SPLINE
SPL {X  -162.820, Y  +507.703, Z    +0.000, E1   -49.462, E3 +312953.270}
SPL {X  -162.820, Y  +516.435, Z    +0.000, E1   -49.526, E3 +312968.239}
SPL {X  -162.820, Y  +523.383, Z    +0.000, E1   -49.407, E3 +312981.426}
SPL {X  -162.820, Y  +532.283, Z    +0.000, E1   -49.462, E3 +312997.028}
SPL {X  -162.820, Y  +541.471, Z    +0.000, E1   -49.456, E3 +313013.407}
SPL {X  -162.820, Y  +548.933, Z    +0.000, E1   -49.456, E3 +313026.595}
SPL {X  -162.820, Y  +553.997, Z    +0.000, E1   -49.325, E3 +313036.399}
SPL {X  -162.820, Y  +562.346, Z    +0.000, E1   -49.498, E3 +313050.461}
SPL {X  -162.820, Y  +570.444, Z    +0.000, E1   -49.421, E3 +313065.208}
SPL {X  -162.820, Y  +577.429, Z    +0.000, E1   -49.474, E3 +313077.322}
SPL {X  -162.820, Y  +585.965, Z    +0.000, E1   -49.447, E3 +313092.896}
SPL {X  -162.820, Y  +594.192, Z    +0.000, E1   -49.325, E3 +313108.139}
SPL {X  -162.820, Y  +600.267, Z    +0.000, E1   -49.443, E3 +313118.228}
SPL {X  -162.820, Y  +606.218, Z    +0.000, E1   -49.464, E3 +313128.775}
SPL {X  -162.820, Y  +612.538, Z    +0.000, E1   -49.488, E3 +313139.826}
SPL {X  -162.820, Y  +617.738, Z    +0.000, E1   -49.301, E3 +313150.262}
SPL {X  -162.820, Y  +624.265, Z    +0.000, E1   -49.443, E3 +313161.057}
SPL {X  -162.820, Y  +630.226, Z    +0.000, E1   -49.472, E3 +313171.505}
SPL {X  -162.820, Y  +635.239, Z    +0.000, E1   -49.373, E3 +313181.001}
SPL {X  -162.820, Y  +641.207, Z    +0.000, E1   -49.420, E3 +313191.469}
SPL {X  -162.820, Y  +649.864, Z    +0.000, E1   -49.433, E3 +313206.947}
SPL {X  -162.820, Y  +658.147, Z    +0.000, E1   -49.491, E3 +313221.214}
SPL {X  -162.820, Y  +663.916, Z    +0.000, E1   -49.371, E3 +313232.204}
SPL {X  -162.820, Y  +669.755, Z    +0.000, E1   -49.387, E3 +313242.529}
SPL {X  -162.807, Y  +675.597, Z    +0.000, E1   -49.472, E3 +313252.431}
SPL {X  -162.632, Y  +681.322, Z    +0.000, E1   -49.345, E3 +313263.443}
SPL {X  -162.228, Y  +687.372, Z    +0.000, E1   -49.294, E3 +313274.529}
SPL {X  -161.723, Y  +692.372, Z    +0.000, E1   -49.172, E3 +313284.159}
SPL {X  -161.009, Y  +697.714, Z    +0.000, E1   -49.214, E3 +313293.444}
SPL {X  -160.313, Y  +701.965, Z    +0.000, E1   -48.932, E3 +313302.656}
SPL {X  -158.980, Y  +708.651, Z    +0.000, E1   -48.774, E3 +313315.696}
SPL {X  -157.477, Y  +714.869, Z    +0.000, E1   -48.424, E3 +313328.571}
SPL {X  -156.071, Y  +719.891, Z    +0.000, E1   -48.264, E3 +313338.447}
SPL {X  -154.661, Y  +724.395, Z    +0.000, E1   -47.951, E3 +313348.129}
SPL {X  -153.094, Y  +728.931, Z    +0.000, E1   -47.705, E3 +313357.565}
SPL {X  -151.300, Y  +733.655, Z    +0.000, E1   -47.339, E3 +313367.874}
SPL {X  -145.669, Y  +746.239, Z    +0.000, E1   -50.198, E3 +313374.650}
SPL {X  -135.559, Y  +763.690, Z    +0.000, E1   -44.340, E3 +313461.445}
ENDSPLINE

SPLINE
SPL {X  -153.801, Y  +726.938, Z    +0.000, E1   -29.643, E3 +313530.158}
SPL {X  -160.383, Y  +701.564, Z    +0.000, E1   -18.145, E3 +313538.297}
SPL {X  -162.078, Y  +689.023, Z    +0.000, E1   -11.510, E3 +313537.835}
SPL {X  -162.685, Y  +680.136, Z    +0.000, E1    -6.379, E3 +313538.124}
SPL {X  -162.820, Y  +672.919, Z    +0.000, E1    -1.752, E3 +313538.163}
SPL {X  -162.820, Y  +667.861, Z    +0.000, E1    +2.254, E3 +313537.964}
SPL {X  -162.820, Y  +662.755, Z    +0.000, E1    +7.521, E3 +313538.005}
SPL {X  -162.820, Y  +657.537, Z    +0.000, E1   +13.540, E3 +313537.674}
SPL {X  -162.820, Y  +650.460, Z    +0.000, E1   +22.200, E3 +313537.105}
SPL {X  -162.820, Y  +637.843, Z    +0.000, E1   +35.051, E3 +313539.182}
SPL {X  -162.820, Y  +595.072, Z    +0.000, E1   +53.652, E3 +313559.902}
SPL {X  -162.820, Y  +560.706, Z    +0.000, E1   +50.482, E3 +313620.811}
ENDSPLINE

SPLINE
SPL {X  -162.820, Y  +560.978, Z    +0.000, E1   +48.448, E3 +313632.897}
ENDSPLINE

SPLINE
SPL {X  -162.820, Y  +552.125, Z    +0.000, E1   +48.477, E3 +313649.002}
SPL {X  -162.820, Y  +545.800, Z    +0.000, E1   +48.334, E3 +313661.443}
SPL {X  -162.820, Y  +540.645, Z    +0.000, E1   +48.364, E3 +313670.794}
SPL {X  -162.820, Y  +534.689, Z    +0.000, E1   +48.295, E3 +313682.343}
SPL {X  -162.820, Y  +526.053, Z    +0.000, E1   +48.382, E3 +313697.918}
SPL {X  -162.820, Y  +516.130, Z    +0.000, E1   +48.458, E3 +313715.876}
SPL {X  -162.820, Y  +508.282, Z    +0.000, E1   +48.307, E3 +313731.131}
SPL {X  -162.820, Y  +502.890, Z    +0.000, E1   +48.309, E3 +313741.058}
ENDSPLINE

SPLINE
SPL {X  -162.820, Y  +517.326, Z    +0.000, E1   +41.232, E3 +313753.322}
ENDSPLINE

SPLINE
SPL {X  -162.820, Y  +509.871, Z    +0.000, E1   +42.115, E3 +313765.423}
SPL {X  -162.820, Y  +504.481, Z    +0.000, E1   +42.725, E3 +313774.088}
SPL {X  -162.820, Y  +496.780, Z    +0.000, E1   +43.573, E3 +313786.255}
SPL {X  -162.820, Y  +488.962, Z    +0.000, E1   +44.342, E3 +313798.523}
SPL {X  -162.820, Y  +481.373, Z    +0.000, E1   +45.107, E3 +313810.007}
SPL {X  -162.820, Y  +473.909, Z    +0.000, E1   +45.743, E3 +313821.520}
SPL {X  -162.820, Y  +465.836, Z    +0.000, E1   +46.727, E3 +313831.810}
SPL {X  -162.820, Y  +457.217, Z    +0.000, E1   +47.671, E3 +313842.848}
SPL {X  -162.820, Y  +449.104, Z    +0.000, E1   +48.459, E3 +313853.317}
SPL {X  -162.820, Y  +438.072, Z    +0.000, E1   +49.432, E3 +313867.672}
SPL {X  -162.820, Y  +428.488, Z    +0.000, E1   +49.830, E3 +313882.107}
SPL {X  -162.820, Y  +423.062, Z    +0.000, E1   +49.728, E3 +313892.250}
SPL {X  -162.820, Y  +416.560, Z    +0.000, E1   +49.816, E3 +313903.231}
SPL {X  -162.820, Y  +410.559, Z    +0.000, E1   +49.727, E3 +313914.286}
SPL {X  -162.820, Y  +405.170, Z    +0.000, E1   +49.772, E3 +313923.488}
SPL {X  -162.820, Y  +398.766, Z    +0.000, E1   +49.793, E3 +313934.775}
SPL {X  -162.820, Y  +391.831, Z    +0.000, E1   +49.801, E3 +313946.821}
SPL {X  -162.820, Y  +386.334, Z    +0.000, E1   +49.739, E3 +313956.910}
SPL {X  -162.801, Y  +377.981, Z    +0.000, E1   +49.798, E3 +313971.431}
SPL {X  -162.314, Y  +367.677, Z    +0.000, E1   +49.734, E3 +313990.071}
SPL {X  -161.359, Y  +358.734, Z    +0.000, E1   +49.535, E3 +314006.855}
SPL {X  -160.051, Y  +350.597, Z    +0.000, E1   +49.332, E3 +314022.465}
SPL {X  -158.863, Y  +344.823, Z    +0.000, E1   +49.020, E3 +314034.193}
SPL {X  -157.695, Y  +339.971, Z    +0.000, E1   +48.934, E3 +314043.289}
SPL {X  -156.136, Y  +334.326, Z    +0.000, E1   +48.578, E3 +314055.256}
SPL {X  -154.561, Y  +329.302, Z    +0.000, E1   +48.290, E3 +314065.586}
SPL {X  -152.787, Y  +324.229, Z    +0.000, E1   +47.981, E3 +314076.276}
SPL {X  -150.789, Y  +319.074, Z    +0.000, E1   +47.585, E3 +314087.299}
SPL {X  -145.123, Y  +306.679, Z    +0.000, E1   +50.518, E3 +314093.196}
SPL {X  -135.207, Y  +289.783, Z    +0.000, E1   +44.101, E3 +314186.711}
ENDSPLINE

SPLINE
SPL {X  -154.528, Y  +329.203, Z    +0.000, E1   +28.834, E3 +314257.072}
SPL {X  -160.380, Y  +352.419, Z    +0.000, E1   +18.163, E3 +314261.432}
SPL {X  -162.408, Y  +368.921, Z    +0.000, E1    +9.337, E3 +314260.182}
SPL {X  -162.817, Y  +379.558, Z    +0.000, E1    +2.744, E3 +314260.572}
SPL {X  -162.820, Y  +383.077, Z    +0.000, E1    +0.110, E3 +314260.968}
SPL {X  -162.820, Y  +386.028, Z    +0.000, E1    -2.328, E3 +314260.291}
SPL {X  -162.820, Y  +389.792, Z    +0.000, E1    -6.211, E3 +314260.223}
SPL {X  -162.820, Y  +394.068, Z    +0.000, E1   -11.043, E3 +314260.340}
SPL {X  -162.820, Y  +398.921, Z    +0.000, E1   -16.945, E3 +314260.393}
SPL {X  -162.820, Y  +406.317, Z    +0.000, E1   -26.128, E3 +314259.206}
SPL {X  -162.820, Y  +413.297, Z    +0.000, E1   -33.931, E3 +314259.195}
SPL {X  -162.820, Y  +446.299, Z    +0.000, E1   -49.360, E3 +314279.705}
SPL {X  -162.820, Y  +502.427, Z    +0.000, E1   -53.345, E3 +314342.691}
ENDSPLINE

SPLINE
SPL {X  -162.820, Y  +494.458, Z    +0.000, E1   -49.332, E3 +314353.223}
ENDSPLINE

SPLINE
SPL {X  -162.820, Y  +499.429, Z    +0.000, E1   -49.453, E3 +314361.432}
SPL {X  -162.820, Y  +507.703, Z    +0.000, E1   -49.462, E3 +314376.347}
SPL {X  -162.820, Y  +516.435, Z    +0.000, E1   -49.526, E3 +314391.316}
SPL {X  -162.820, Y  +522.095, Z    +0.000, E1   -49.420, E3 +314402.013}
SPL {X  -162.820, Y  +529.397, Z    +0.000, E1   -49.440, E3 +314415.021}
SPL {X  -162.820, Y  +535.099, Z    +0.000, E1   -49.339, E3 +314425.639}
SPL {X  -162.820, Y  +541.471, Z    +0.000, E1   -49.456, E3 +314436.484}
SPL {X  -162.820, Y  +548.933, Z    +0.000, E1   -49.456, E3 +314449.672}
SPL {X  -162.820, Y  +553.997, Z    +0.000, E1   -49.325, E3 +314459.476}
SPL {X  -162.820, Y  +560.268, Z    +0.000, E1   -49.531, E3 +314469.434}
SPL {X  -162.820, Y  +564.590, Z    +0.000, E1   -49.361, E3 +314478.133}
SPL {X  -162.820, Y  +570.444, Z    +0.000, E1   -49.421, E3 +314488.285}
SPL {X  -162.820, Y  +577.429, Z    +0.000, E1   -49.474, E3 +314500.399}
SPL {X  -162.820, Y  +582.387, Z    +0.000, E1   -49.269, E3 +314510.420}
SPL {X  -162.820, Y  +588.456, Z    +0.000, E1   -49.496, E3 +314519.935}
SPL {X  -162.820, Y  +594.192, Z    +0.000, E1   -49.325, E3 +314531.216}
SPL {X  -162.820, Y  +600.267, Z    +0.000, E1   -49.443, E3 +314541.305}
SPL {X  -162.820, Y  +606.218, Z    +0.000, E1   -49.464, E3 +314551.851}
SPL {X  -162.820, Y  +612.538, Z    +0.000, E1   -49.488, E3 +314562.902}
SPL {X  -162.820, Y  +617.738, Z    +0.000, E1   -49.301, E3 +314573.339}
SPL {X  -162.820, Y  +624.265, Z    +0.000, E1   -49.443, E3 +314584.134}
SPL {X  -162.820, Y  +630.226, Z    +0.000, E1   -49.472, E3 +314594.582}
SPL {X  -162.820, Y  +635.239, Z    +0.000, E1   -49.373, E3 +314604.077}
SPL {X  -162.820, Y  +641.207, Z    +0.000, E1   -49.420, E3 +314614.546}
SPL {X  -162.820, Y  +649.864, Z    +0.000, E1   -49.433, E3 +314630.024}
SPL {X  -162.820, Y  +658.147, Z    +0.000, E1   -49.491, E3 +314644.291}
SPL {X  -162.820, Y  +663.916, Z    +0.000, E1   -49.371, E3 +314655.281}
SPL {X  -162.820, Y  +669.755, Z    +0.000, E1   -49.387, E3 +314665.606}
SPL {X  -162.807, Y  +675.597, Z    +0.000, E1   -49.472, E3 +314675.508}
SPL {X  -162.632, Y  +681.322, Z    +0.000, E1   -49.345, E3 +314686.520}
SPL {X  -162.228, Y  +687.372, Z    +0.000, E1   -49.294, E3 +314697.606}
SPL {X  -161.723, Y  +692.372, Z    +0.000, E1   -49.172, E3 +314707.236}
SPL {X  -161.009, Y  +697.714, Z    +0.000, E1   -49.214, E3 +314716.521}
SPL {X  -160.313, Y  +701.965, Z    +0.000, E1   -48.932, E3 +314725.733}
SPL {X  -158.980, Y  +708.651, Z    +0.000, E1   -48.774, E3 +314738.773}
SPL {X  -157.477, Y  +714.869, Z    +0.000, E1   -48.424, E3 +314751.648}
SPL {X  -156.071, Y  +719.891, Z    +0.000, E1   -48.264, E3 +314761.524}
SPL {X  -154.661, Y  +724.395, Z    +0.000, E1   -47.951, E3 +314771.206}
SPL {X  -153.094, Y  +728.931, Z    +0.000, E1   -47.705, E3 +314780.642}
SPL {X  -151.300, Y  +733.655, Z    +0.000, E1   -47.339, E3 +314790.951}
SPL {X  -145.669, Y  +746.239, Z    +0.000, E1   -50.198, E3 +314797.727}
SPL {X  -135.084, Y  +764.399, Z    +0.000, E1   -44.787, E3 +314880.631}
ENDSPLINE

SPLINE
SPL {X  -153.038, Y  +729.086, Z    +0.000, E1   -30.522, E3 +314951.338}
SPL {X  -160.383, Y  +701.564, Z    +0.000, E1   -18.145, E3 +314961.374}
SPL {X  -162.078, Y  +689.023, Z    +0.000, E1   -11.510, E3 +314960.912}
SPL {X  -162.685, Y  +680.136, Z    +0.000, E1    -6.379, E3 +314961.201}
SPL {X  -162.820, Y  +672.919, Z    +0.000, E1    -1.752, E3 +314961.240}
SPL {X  -162.820, Y  +667.861, Z    +0.000, E1    +2.254, E3 +314961.041}
SPL {X  -162.820, Y  +662.755, Z    +0.000, E1    +7.521, E3 +314961.082}
SPL {X  -162.820, Y  +657.537, Z    +0.000, E1   +13.540, E3 +314960.751}
SPL {X  -162.820, Y  +650.460, Z    +0.000, E1   +22.200, E3 +314960.182}
SPL {X  -162.820, Y  +637.843, Z    +0.000, E1   +35.051, E3 +314962.259}
SPL {X  -162.820, Y  +595.072, Z    +0.000, E1   +53.652, E3 +314982.979}
SPL {X  -162.820, Y  +560.706, Z    +0.000, E1   +50.482, E3 +315043.888}
ENDSPLINE

SPLINE
SPL {X  -162.820, Y  +560.978, Z    +0.000, E1   +48.448, E3 +315055.974}
ENDSPLINE

SPLINE
SPL {X  -162.820, Y  +552.125, Z    +0.000, E1   +48.477, E3 +315072.078}
SPL {X  -162.820, Y  +545.800, Z    +0.000, E1   +48.334, E3 +315084.520}
SPL {X  -162.820, Y  +540.645, Z    +0.000, E1   +48.364, E3 +315093.871}
SPL {X  -162.820, Y  +534.689, Z    +0.000, E1   +48.295, E3 +315105.420}
SPL {X  -162.820, Y  +526.053, Z    +0.000, E1   +48.382, E3 +315120.995}
SPL {X  -162.820, Y  +516.130, Z    +0.000, E1   +48.458, E3 +315138.953}
SPL {X  -162.820, Y  +508.282, Z    +0.000, E1   +48.307, E3 +315154.208}
SPL {X  -162.820, Y  +502.890, Z    +0.000, E1   +48.309, E3 +315164.135}
ENDSPLINE

SPLINE
SPL {X  -162.820, Y  +517.326, Z    +0.000, E1   +41.232, E3 +315176.399}
ENDSPLINE

SPLINE
SPL {X  -162.820, Y  +509.871, Z    +0.000, E1   +42.115, E3 +315188.500}
SPL {X  -162.820, Y  +504.481, Z    +0.000, E1   +42.725, E3 +315197.165}
SPL {X  -162.820, Y  +496.780, Z    +0.000, E1   +43.573, E3 +315209.332}
SPL {X  -162.820, Y  +488.962, Z    +0.000, E1   +44.342, E3 +315221.600}
SPL {X  -162.820, Y  +481.373, Z    +0.000, E1   +45.107, E3 +315233.084}
SPL {X  -162.820, Y  +473.909, Z    +0.000, E1   +45.743, E3 +315244.596}
SPL {X  -162.820, Y  +465.836, Z    +0.000, E1   +46.727, E3 +315254.887}
SPL {X  -162.820, Y  +457.217, Z    +0.000, E1   +47.671, E3 +315265.925}
SPL {X  -162.820, Y  +449.104, Z    +0.000, E1   +48.459, E3 +315276.394}
SPL {X  -162.820, Y  +438.072, Z    +0.000, E1   +49.432, E3 +315290.749}
SPL {X  -162.820, Y  +428.488, Z    +0.000, E1   +49.830, E3 +315305.184}
SPL {X  -162.820, Y  +423.062, Z    +0.000, E1   +49.728, E3 +315315.327}
SPL {X  -162.820, Y  +416.560, Z    +0.000, E1   +49.816, E3 +315326.307}
SPL {X  -162.820, Y  +410.559, Z    +0.000, E1   +49.727, E3 +315337.363}
SPL {X  -162.820, Y  +405.170, Z    +0.000, E1   +49.772, E3 +315346.565}
SPL {X  -162.820, Y  +398.766, Z    +0.000, E1   +49.793, E3 +315357.852}
SPL {X  -162.820, Y  +391.831, Z    +0.000, E1   +49.801, E3 +315369.898}
SPL {X  -162.820, Y  +386.334, Z    +0.000, E1   +49.739, E3 +315379.986}
SPL {X  -162.801, Y  +377.981, Z    +0.000, E1   +49.798, E3 +315394.508}
SPL {X  -162.314, Y  +367.677, Z    +0.000, E1   +49.734, E3 +315413.148}
SPL {X  -161.359, Y  +358.734, Z    +0.000, E1   +49.535, E3 +315429.932}
SPL {X  -160.051, Y  +350.597, Z    +0.000, E1   +49.332, E3 +315445.542}
SPL {X  -158.863, Y  +344.823, Z    +0.000, E1   +49.020, E3 +315457.270}
SPL {X  -157.695, Y  +339.971, Z    +0.000, E1   +48.934, E3 +315466.366}
SPL {X  -156.136, Y  +334.326, Z    +0.000, E1   +48.578, E3 +315478.332}
SPL {X  -154.561, Y  +329.302, Z    +0.000, E1   +48.290, E3 +315488.663}
SPL {X  -152.787, Y  +324.229, Z    +0.000, E1   +47.981, E3 +315499.353}
SPL {X  -150.789, Y  +319.074, Z    +0.000, E1   +47.585, E3 +315510.376}
SPL {X  -145.123, Y  +306.679, Z    +0.000, E1   +50.518, E3 +315516.273}
SPL {X  -135.207, Y  +289.783, Z    +0.000, E1   +44.101, E3 +315609.788}
ENDSPLINE

SPLINE
SPL {X  -154.528, Y  +329.203, Z    +0.000, E1   +28.834, E3 +315680.149}
SPL {X  -160.380, Y  +352.419, Z    +0.000, E1   +18.163, E3 +315684.509}
SPL {X  -162.408, Y  +368.921, Z    +0.000, E1    +9.337, E3 +315683.259}
SPL {X  -162.817, Y  +379.558, Z    +0.000, E1    +2.744, E3 +315683.649}
SPL {X  -162.820, Y  +383.077, Z    +0.000, E1    +0.110, E3 +315684.045}
SPL {X  -162.820, Y  +386.028, Z    +0.000, E1    -2.328, E3 +315683.368}
SPL {X  -162.820, Y  +389.792, Z    +0.000, E1    -6.211, E3 +315683.300}
SPL {X  -162.820, Y  +394.068, Z    +0.000, E1   -11.043, E3 +315683.417}
SPL {X  -162.820, Y  +398.921, Z    +0.000, E1   -16.945, E3 +315683.470}
SPL {X  -162.820, Y  +406.317, Z    +0.000, E1   -26.128, E3 +315682.283}
SPL {X  -162.820, Y  +413.297, Z    +0.000, E1   -33.931, E3 +315682.272}
SPL {X  -162.820, Y  +446.299, Z    +0.000, E1   -49.360, E3 +315702.782}
SPL {X  -162.820, Y  +502.427, Z    +0.000, E1   -53.345, E3 +315765.768}
ENDSPLINE

SPLINE
SPL {X  -162.820, Y  +494.458, Z    +0.000, E1   -49.332, E3 +315776.300}
ENDSPLINE

SPLINE
SPL {X  -162.820, Y  +499.429, Z    +0.000, E1   -49.453, E3 +315784.509}
SPL {X  -162.820, Y  +507.703, Z    +0.000, E1   -49.462, E3 +315799.424}
SPL {X  -162.820, Y  +516.435, Z    +0.000, E1   -49.526, E3 +315814.393}
SPL {X  -162.820, Y  +522.095, Z    +0.000, E1   -49.420, E3 +315825.090}
SPL {X  -162.820, Y  +529.397, Z    +0.000, E1   -49.440, E3 +315838.098}
SPL {X  -162.820, Y  +535.099, Z    +0.000, E1   -49.339, E3 +315848.716}
SPL {X  -162.820, Y  +541.471, Z    +0.000, E1   -49.456, E3 +315859.560}
SPL {X  -162.820, Y  +548.933, Z    +0.000, E1   -49.456, E3 +315872.749}
SPL {X  -162.820, Y  +553.997, Z    +0.000, E1   -49.325, E3 +315882.553}
SPL {X  -162.820, Y  +560.268, Z    +0.000, E1   -49.531, E3 +315892.511}
SPL {X  -162.820, Y  +564.590, Z    +0.000, E1   -49.361, E3 +315901.210}
SPL {X  -162.820, Y  +570.444, Z    +0.000, E1   -49.421, E3 +315911.362}
SPL {X  -162.820, Y  +577.429, Z    +0.000, E1   -49.474, E3 +315923.476}
SPL {X  -162.820, Y  +582.387, Z    +0.000, E1   -49.269, E3 +315933.497}
SPL {X  -162.820, Y  +588.456, Z    +0.000, E1   -49.496, E3 +315943.012}
SPL {X  -162.820, Y  +594.192, Z    +0.000, E1   -49.325, E3 +315954.293}
SPL {X  -162.820, Y  +600.267, Z    +0.000, E1   -49.443, E3 +315964.382}
SPL {X  -162.820, Y  +606.218, Z    +0.000, E1   -49.464, E3 +315974.928}
SPL {X  -162.820, Y  +612.538, Z    +0.000, E1   -49.488, E3 +315985.979}
SPL {X  -162.820, Y  +617.738, Z    +0.000, E1   -49.301, E3 +315996.416}
SPL {X  -162.820, Y  +624.265, Z    +0.000, E1   -49.443, E3 +316007.211}
SPL {X  -162.820, Y  +630.226, Z    +0.000, E1   -49.472, E3 +316017.659}
SPL {X  -162.820, Y  +635.239, Z    +0.000, E1   -49.373, E3 +316027.154}
SPL {X  -162.820, Y  +641.207, Z    +0.000, E1   -49.420, E3 +316037.623}
SPL {X  -162.820, Y  +649.864, Z    +0.000, E1   -49.433, E3 +316053.101}
SPL {X  -162.820, Y  +658.147, Z    +0.000, E1   -49.491, E3 +316067.368}
SPL {X  -162.820, Y  +663.916, Z    +0.000, E1   -49.371, E3 +316078.358}
SPL {X  -162.820, Y  +669.755, Z    +0.000, E1   -49.387, E3 +316088.683}
SPL {X  -162.807, Y  +675.597, Z    +0.000, E1   -49.472, E3 +316098.585}
SPL {X  -162.632, Y  +681.322, Z    +0.000, E1   -49.345, E3 +316109.596}
SPL {X  -162.228, Y  +687.372, Z    +0.000, E1   -49.294, E3 +316120.683}
SPL {X  -161.723, Y  +692.372, Z    +0.000, E1   -49.172, E3 +316130.313}
SPL {X  -161.009, Y  +697.714, Z    +0.000, E1   -49.214, E3 +316139.598}
SPL {X  -160.313, Y  +701.965, Z    +0.000, E1   -48.932, E3 +316148.810}
SPL {X  -158.980, Y  +708.651, Z    +0.000, E1   -48.774, E3 +316161.850}
SPL {X  -157.477, Y  +714.869, Z    +0.000, E1   -48.424, E3 +316174.725}
SPL {X  -156.071, Y  +719.891, Z    +0.000, E1   -48.264, E3 +316184.601}
SPL {X  -154.661, Y  +724.395, Z    +0.000, E1   -47.951, E3 +316194.282}
SPL {X  -153.094, Y  +728.931, Z    +0.000, E1   -47.705, E3 +316203.719}
SPL {X  -151.300, Y  +733.655, Z    +0.000, E1   -47.339, E3 +316214.028}
SPL {X  -145.669, Y  +746.239, Z    +0.000, E1   -50.198, E3 +316220.804}
SPL {X  -135.084, Y  +764.399, Z    +0.000, E1   -44.787, E3 +316303.708}
ENDSPLINE

SPLINE
SPL {X  -153.038, Y  +729.086, Z    +0.000, E1   -30.522, E3 +316374.415}
SPL {X  -160.383, Y  +701.564, Z    +0.000, E1   -18.145, E3 +316384.451}
SPL {X  -162.078, Y  +689.023, Z    +0.000, E1   -11.510, E3 +316383.989}
SPL {X  -162.685, Y  +680.136, Z    +0.000, E1    -6.379, E3 +316384.278}
SPL {X  -162.820, Y  +672.919, Z    +0.000, E1    -1.752, E3 +316384.317}
SPL {X  -162.820, Y  +667.861, Z    +0.000, E1    +2.254, E3 +316384.118}
SPL {X  -162.820, Y  +662.755, Z    +0.000, E1    +7.521, E3 +316384.159}
SPL {X  -162.820, Y  +657.537, Z    +0.000, E1   +13.540, E3 +316383.828}
SPL {X  -162.820, Y  +650.460, Z    +0.000, E1   +22.200, E3 +316383.259}
SPL {X  -162.820, Y  +637.843, Z    +0.000, E1   +35.051, E3 +316385.336}
SPL {X  -162.820, Y  +595.072, Z    +0.000, E1   +53.652, E3 +316406.056}
SPL {X  -162.820, Y  +560.706, Z    +0.000, E1   +50.482, E3 +316466.965}
ENDSPLINE

SPLINE
SPL {X  -162.820, Y  +560.978, Z    +0.000, E1   +48.448, E3 +316479.051}
ENDSPLINE

SPLINE
SPL {X  -162.820, Y  +552.125, Z    +0.000, E1   +48.477, E3 +316495.155}
SPL {X  -162.820, Y  +545.800, Z    +0.000, E1   +48.334, E3 +316507.597}
SPL {X  -162.820, Y  +540.645, Z    +0.000, E1   +48.364, E3 +316516.948}
SPL {X  -162.820, Y  +534.689, Z    +0.000, E1   +48.295, E3 +316528.497}
SPL {X  -162.820, Y  +526.053, Z    +0.000, E1   +48.382, E3 +316544.072}
SPL {X  -162.820, Y  +516.130, Z    +0.000, E1   +48.458, E3 +316562.030}
SPL {X  -162.820, Y  +508.282, Z    +0.000, E1   +48.307, E3 +316577.285}
SPL {X  -162.820, Y  +502.890, Z    +0.000, E1   +48.309, E3 +316587.212}
ENDSPLINE

SPLINE
SPL {X  -162.820, Y  +517.326, Z    +0.000, E1   +41.232, E3 +316599.476}
ENDSPLINE

SPLINE
SPL {X  -162.820, Y  +509.871, Z    +0.000, E1   +42.115, E3 +316611.577}
SPL {X  -162.820, Y  +504.481, Z    +0.000, E1   +42.725, E3 +316620.242}
SPL {X  -162.820, Y  +496.780, Z    +0.000, E1   +43.573, E3 +316632.409}
SPL {X  -162.820, Y  +488.962, Z    +0.000, E1   +44.342, E3 +316644.676}
SPL {X  -162.820, Y  +481.373, Z    +0.000, E1   +45.107, E3 +316656.161}
SPL {X  -162.820, Y  +473.909, Z    +0.000, E1   +45.743, E3 +316667.673}
SPL {X  -162.820, Y  +465.836, Z    +0.000, E1   +46.727, E3 +316677.964}
SPL {X  -162.820, Y  +457.217, Z    +0.000, E1   +47.671, E3 +316689.002}
SPL {X  -162.820, Y  +449.104, Z    +0.000, E1   +48.459, E3 +316699.471}
SPL {X  -162.820, Y  +438.072, Z    +0.000, E1   +49.432, E3 +316713.826}
SPL {X  -162.820, Y  +428.488, Z    +0.000, E1   +49.830, E3 +316728.261}
SPL {X  -162.820, Y  +423.062, Z    +0.000, E1   +49.728, E3 +316738.403}
SPL {X  -162.820, Y  +416.560, Z    +0.000, E1   +49.816, E3 +316749.384}
SPL {X  -162.820, Y  +410.559, Z    +0.000, E1   +49.727, E3 +316760.440}
SPL {X  -162.820, Y  +405.170, Z    +0.000, E1   +49.772, E3 +316769.642}
SPL {X  -162.820, Y  +398.766, Z    +0.000, E1   +49.793, E3 +316780.929}
SPL {X  -162.820, Y  +391.831, Z    +0.000, E1   +49.801, E3 +316792.975}
SPL {X  -162.820, Y  +386.334, Z    +0.000, E1   +49.739, E3 +316803.063}
SPL {X  -162.801, Y  +377.981, Z    +0.000, E1   +49.798, E3 +316817.585}
SPL {X  -162.314, Y  +367.677, Z    +0.000, E1   +49.734, E3 +316836.225}
SPL {X  -161.359, Y  +358.734, Z    +0.000, E1   +49.535, E3 +316853.008}
SPL {X  -160.051, Y  +350.597, Z    +0.000, E1   +49.332, E3 +316868.619}
SPL {X  -158.863, Y  +344.823, Z    +0.000, E1   +49.020, E3 +316880.347}
SPL {X  -157.695, Y  +339.971, Z    +0.000, E1   +48.934, E3 +316889.443}
SPL {X  -156.136, Y  +334.326, Z    +0.000, E1   +48.578, E3 +316901.409}
SPL {X  -154.561, Y  +329.302, Z    +0.000, E1   +48.290, E3 +316911.740}
SPL {X  -152.787, Y  +324.229, Z    +0.000, E1   +47.981, E3 +316922.430}
SPL {X  -150.789, Y  +319.074, Z    +0.000, E1   +47.585, E3 +316933.453}
SPL {X  -145.123, Y  +306.679, Z    +0.000, E1   +50.518, E3 +316939.350}
SPL {X  -135.207, Y  +289.783, Z    +0.000, E1   +44.101, E3 +317032.865}
ENDSPLINE

SPLINE
SPL {X  -154.528, Y  +329.203, Z    +0.000, E1   +28.834, E3 +317103.226}
SPL {X  -160.380, Y  +352.419, Z    +0.000, E1   +18.163, E3 +317107.586}
SPL {X  -162.149, Y  +365.734, Z    +0.000, E1   +11.090, E3 +317106.195}
SPL {X  -162.754, Y  +375.862, Z    +0.000, E1    +5.134, E3 +317107.031}
SPL {X  -162.820, Y  +382.085, Z    +0.000, E1    +0.928, E3 +317106.720}
SPL {X  -162.820, Y  +386.028, Z    +0.000, E1    -2.328, E3 +317106.445}
SPL {X  -162.820, Y  +389.792, Z    +0.000, E1    -6.211, E3 +317106.377}
SPL {X  -162.820, Y  +394.068, Z    +0.000, E1   -11.043, E3 +317106.493}
SPL {X  -162.820, Y  +398.921, Z    +0.000, E1   -16.945, E3 +317106.547}
SPL {X  -162.820, Y  +409.049, Z    +0.000, E1   -29.128, E3 +317105.356}
SPL {X  -162.820, Y  +446.299, Z    +0.000, E1   -49.360, E3 +317125.859}
SPL {X  -162.820, Y  +502.427, Z    +0.000, E1   -53.345, E3 +317188.845}
ENDSPLINE

SPLINE
SPL {X  -162.820, Y  +497.758, Z    +0.000, E1   -49.444, E3 +317204.784}
ENDSPLINE

SPLINE
SPL {X  -162.820, Y  +507.703, Z    +0.000, E1   -49.462, E3 +317222.501}
SPL {X  -162.820, Y  +516.435, Z    +0.000, E1   -49.526, E3 +317237.470}
SPL {X  -162.820, Y  +522.095, Z    +0.000, E1   -49.420, E3 +317248.166}
SPL {X  -162.820, Y  +529.397, Z    +0.000, E1   -49.440, E3 +317261.175}
SPL {X  -162.820, Y  +536.932, Z    +0.000, E1   -49.395, E3 +317274.816}
SPL {X  -162.820, Y  +543.021, Z    +0.000, E1   -49.432, E3 +317285.422}
SPL {X  -162.820, Y  +548.933, Z    +0.000, E1   -49.456, E3 +317295.826}
SPL {X  -162.820, Y  +553.997, Z    +0.000, E1   -49.325, E3 +317305.630}
SPL {X  -162.820, Y  +562.346, Z    +0.000, E1   -49.498, E3 +317319.692}
SPL {X  -162.820, Y  +570.444, Z    +0.000, E1   -49.421, E3 +317334.439}
SPL {X  -162.820, Y  +577.429, Z    +0.000, E1   -49.474, E3 +317346.553}
SPL {X  -162.820, Y  +582.387, Z    +0.000, E1   -49.269, E3 +317356.574}
SPL {X  -162.820, Y  +588.456, Z    +0.000, E1   -49.496, E3 +317366.089}
SPL {X  -162.820, Y  +594.192, Z    +0.000, E1   -49.325, E3 +317377.370}
SPL {X  -162.820, Y  +600.267, Z    +0.000, E1   -49.443, E3 +317387.458}
SPL {X  -162.820, Y  +606.218, Z    +0.000, E1   -49.464, E3 +317398.005}
SPL {X  -162.820, Y  +612.538, Z    +0.000, E1   -49.488, E3 +317409.056}
SPL {X  -162.820, Y  +617.738, Z    +0.000, E1   -49.301, E3 +317419.493}
SPL {X  -162.820, Y  +624.265, Z    +0.000, E1   -49.443, E3 +317430.288}
SPL {X  -162.820, Y  +632.551, Z    +0.000, E1   -49.478, E3 +317445.057}
SPL {X  -162.820, Y  +641.207, Z    +0.000, E1   -49.420, E3 +317460.700}
SPL {X  -162.820, Y  +648.011, Z    +0.000, E1   -49.484, E3 +317472.377}
SPL {X  -162.820, Y  +655.976, Z    +0.000, E1   -49.445, E3 +317487.006}
SPL {X  -162.820, Y  +663.916, Z    +0.000, E1   -49.371, E3 +317501.435}
SPL {X  -162.820, Y  +669.755, Z    +0.000, E1   -49.387, E3 +317511.760}
SPL {X  -162.807, Y  +675.597, Z    +0.000, E1   -49.472, E3 +317521.662}
SPL {X  -162.632, Y  +681.322, Z    +0.000, E1   -49.345, E3 +317532.673}
SPL {X  -162.228, Y  +687.372, Z    +0.000, E1   -49.294, E3 +317543.760}
SPL {X  -161.723, Y  +692.372, Z    +0.000, E1   -49.172, E3 +317553.390}
SPL {X  -161.009, Y  +697.714, Z    +0.000, E1   -49.214, E3 +317562.675}
SPL {X  -160.313, Y  +701.965, Z    +0.000, E1   -48.932, E3 +317571.887}
SPL {X  -159.435, Y  +706.528, Z    +0.000, E1   -48.764, E3 +317581.014}
SPL {X  -157.894, Y  +713.249, Z    +0.000, E1   -48.586, E3 +317594.207}
SPL {X  -156.071, Y  +719.891, Z    +0.000, E1   -48.264, E3 +317607.678}
SPL {X  -154.661, Y  +724.395, Z    +0.000, E1   -47.951, E3 +317617.359}
SPL {X  -153.094, Y  +728.931, Z    +0.000, E1   -47.705, E3 +317626.796}
SPL {X  -151.300, Y  +733.655, Z    +0.000, E1   -47.339, E3 +317637.105}
SPL {X  -145.669, Y  +746.239, Z    +0.000, E1   -50.198, E3 +317643.881}
SPL {X  -135.084, Y  +764.399, Z    +0.000, E1   -44.787, E3 +317726.785}
ENDSPLINE

SPLINE
SPL {X  -153.038, Y  +729.086, Z    +0.000, E1   -30.522, E3 +317797.492}
SPL {X  -160.383, Y  +701.564, Z    +0.000, E1   -18.145, E3 +317807.528}
SPL {X  -162.078, Y  +689.023, Z    +0.000, E1   -11.510, E3 +317807.066}
SPL {X  -162.685, Y  +680.136, Z    +0.000, E1    -6.379, E3 +317807.355}
SPL {X  -162.820, Y  +672.919, Z    +0.000, E1    -1.752, E3 +317807.394}
SPL {X  -162.820, Y  +669.270, Z    +0.000, E1    +1.140, E3 +317806.876}
SPL {X  -162.820, Y  +666.754, Z    +0.000, E1    +3.396, E3 +317807.445}
SPL {X  -162.820, Y  +662.755, Z    +0.000, E1    +7.521, E3 +317807.235}
SPL {X  -162.820, Y  +657.537, Z    +0.000, E1   +13.540, E3 +317806.905}
SPL {X  -162.820, Y  +650.460, Z    +0.000, E1   +22.200, E3 +317806.336}
SPL {X  -162.820, Y  +637.843, Z    +0.000, E1   +35.051, E3 +317808.413}
SPL {X  -162.820, Y  +595.072, Z    +0.000, E1   +53.652, E3 +317829.133}
SPL {X  -162.820, Y  +561.831, Z    +0.000, E1   +49.171, E3 +317896.355}
SPL {X  -162.820, Y  +555.289, Z    +0.000, E1   +48.406, E3 +317912.816}
SPL {X  -162.820, Y  +547.003, Z    +0.000, E1   +48.390, E3 +317928.229}
SPL {X  -162.820, Y  +540.645, Z    +0.000, E1   +48.364, E3 +317940.025}
SPL {X  -162.820, Y  +534.689, Z    +0.000, E1   +48.295, E3 +317951.574}
SPL {X  -162.820, Y  +528.564, Z    +0.000, E1   +48.407, E3 +317962.147}
SPL {X  -162.820, Y  +522.157, Z    +0.000, E1   +48.326, E3 +317974.728}
SPL {X  -162.820, Y  +513.750, Z    +0.000, E1   +48.520, E3 +317988.960}
SPL {X  -162.820, Y  +508.282, Z    +0.000, E1   +48.307, E3 +318000.362}
SPL {X  -162.820, Y  +502.890, Z    +0.000, E1   +48.309, E3 +318010.289}
ENDSPLINE

SPLINE
SPL {X  -162.820, Y  +517.326, Z    +0.000, E1   +41.232, E3 +318022.553}
ENDSPLINE

SPLINE
SPL {X  -162.820, Y  +509.871, Z    +0.000, E1   +42.115, E3 +318034.654}
SPL {X  -162.820, Y  +501.934, Z    +0.000, E1   +43.022, E3 +318047.381}
SPL {X  -162.820, Y  +494.356, Z    +0.000, E1   +43.819, E3 +318059.222}
SPL {X  -162.820, Y  +487.058, Z    +0.000, E1   +44.544, E3 +318070.686}
SPL {X  -162.820, Y  +476.193, Z    +0.000, E1   +45.591, E3 +318087.125}
SPL {X  -162.820, Y  +465.836, Z    +0.000, E1   +46.727, E3 +318101.041}
SPL {X  -162.820, Y  +457.217, Z    +0.000, E1   +47.671, E3 +318112.079}
SPL {X  -162.820, Y  +446.677, Z    +0.000, E1   +48.707, E3 +318125.608}
SPL {X  -162.820, Y  +435.978, Z    +0.000, E1   +49.560, E3 +318139.758}
SPL {X  -162.820, Y  +428.488, Z    +0.000, E1   +49.830, E3 +318151.337}
SPL {X  -162.820, Y  +423.062, Z    +0.000, E1   +49.728, E3 +318161.480}
SPL {X  -162.820, Y  +416.560, Z    +0.000, E1   +49.816, E3 +318172.461}
SPL {X  -162.820, Y  +407.996, Z    +0.000, E1   +49.793, E3 +318187.827}
SPL {X  -162.820, Y  +398.766, Z    +0.000, E1   +49.793, E3 +318204.006}
SPL {X  -162.820, Y  +391.831, Z    +0.000, E1   +49.801, E3 +318216.052}
SPL {X  -162.820, Y  +386.334, Z    +0.000, E1   +49.739, E3 +318226.140}
SPL {X  -162.801, Y  +377.981, Z    +0.000, E1   +49.798, E3 +318240.662}
SPL {X  -162.314, Y  +367.677, Z    +0.000, E1   +49.734, E3 +318259.302}
SPL {X  -161.359, Y  +358.734, Z    +0.000, E1   +49.535, E3 +318276.085}
SPL {X  -160.051, Y  +350.597, Z    +0.000, E1   +49.332, E3 +318291.696}
SPL {X  -158.863, Y  +344.823, Z    +0.000, E1   +49.020, E3 +318303.424}
SPL {X  -157.695, Y  +339.971, Z    +0.000, E1   +48.934, E3 +318312.520}
SPL {X  -156.136, Y  +334.326, Z    +0.000, E1   +48.578, E3 +318324.486}
SPL {X  -153.956, Y  +327.511, Z    +0.000, E1   +48.205, E3 +318338.608}
SPL {X  -151.655, Y  +321.245, Z    +0.000, E1   +47.770, E3 +318351.818}
SPL {X  -148.347, Y  +313.391, Z    +0.000, E1   +48.924, E3 +318359.415}
SPL {X  -143.047, Y  +302.732, Z    +0.000, E1   +51.043, E3 +318365.935}
SPL {X  -135.207, Y  +289.783, Z    +0.000, E1   +44.101, E3 +318455.942}
ENDSPLINE

SPLINE
SPL {X  -154.528, Y  +329.203, Z    +0.000, E1   +28.834, E3 +318526.303}
SPL {X  -160.380, Y  +352.419, Z    +0.000, E1   +18.163, E3 +318530.663}
SPL {X  -162.149, Y  +365.734, Z    +0.000, E1   +11.090, E3 +318529.272}
SPL {X  -162.754, Y  +375.862, Z    +0.000, E1    +5.134, E3 +318530.108}
SPL {X  -162.820, Y  +381.027, Z    +0.000, E1    +1.647, E3 +318529.368}
SPL {X  -162.820, Y  +384.383, Z    +0.000, E1    -0.869, E3 +318529.773}
SPL {X  -162.820, Y  +388.871, Z    +0.000, E1    -5.151, E3 +318529.479}
SPL {X  -162.820, Y  +394.068, Z    +0.000, E1   -11.043, E3 +318529.570}
SPL {X  -162.820, Y  +398.921, Z    +0.000, E1   -16.945, E3 +318529.624}
SPL {X  -162.820, Y  +406.317, Z    +0.000, E1   -26.128, E3 +318528.437}
SPL {X  -162.820, Y  +413.297, Z    +0.000, E1   -33.931, E3 +318528.426}
SPL {X  -162.820, Y  +446.299, Z    +0.000, E1   -49.360, E3 +318548.936}
SPL {X  -162.820, Y  +502.427, Z    +0.000, E1   -53.345, E3 +318611.921}
ENDSPLINE

SPLINE
SPL {X  -162.820, Y  +494.458, Z    +0.000, E1   -49.332, E3 +318622.454}
ENDSPLINE

SPLINE
SPL {X  -162.820, Y  +499.429, Z    +0.000, E1   -49.453, E3 +318630.663}
SPL {X  -162.820, Y  +505.173, Z    +0.000, E1   -49.386, E3 +318641.319}
SPL {X  -162.820, Y  +510.642, Z    +0.000, E1   -49.447, E3 +318650.669}
SPL {X  -162.820, Y  +516.435, Z    +0.000, E1   -49.526, E3 +318660.547}
SPL {X  -162.820, Y  +523.383, Z    +0.000, E1   -49.407, E3 +318673.734}
SPL {X  -162.820, Y  +532.283, Z    +0.000, E1   -49.462, E3 +318689.336}
SPL {X  -162.820, Y  +541.471, Z    +0.000, E1   -49.456, E3 +318705.714}
SPL {X  -162.820, Y  +548.933, Z    +0.000, E1   -49.456, E3 +318718.903}
SPL {X  -162.820, Y  +553.997, Z    +0.000, E1   -49.325, E3 +318728.707}
SPL {X  -162.820, Y  +560.268, Z    +0.000, E1   -49.531, E3 +318738.664}
SPL {X  -162.820, Y  +564.590, Z    +0.000, E1   -49.361, E3 +318747.364}
SPL {X  -162.820, Y  +570.444, Z    +0.000, E1   -49.421, E3 +318757.516}
SPL {X  -162.820, Y  +577.429, Z    +0.000, E1   -49.474, E3 +318769.630}
SPL {X  -162.820, Y  +585.965, Z    +0.000, E1   -49.447, E3 +318785.204}
SPL {X  -162.820, Y  +594.192, Z    +0.000, E1   -49.325, E3 +318800.447}
SPL {X  -162.820, Y  +600.267, Z    +0.000, E1   -49.443, E3 +318810.535}
SPL {X  -162.820, Y  +606.218, Z    +0.000, E1   -49.464, E3 +318821.082}
SPL {X  -162.820, Y  +612.538, Z    +0.000, E1   -49.488, E3 +318832.133}
SPL {X  -162.820, Y  +617.738, Z    +0.000, E1   -49.301, E3 +318842.570}
SPL {X  -162.820, Y  +624.265, Z    +0.000, E1   -49.443, E3 +318853.365}
SPL {X  -162.820, Y  +630.226, Z    +0.000, E1   -49.472, E3 +318863.813}
SPL {X  -162.820, Y  +635.239, Z    +0.000, E1   -49.373, E3 +318873.308}
SPL {X  -162.820, Y  +641.207, Z    +0.000, E1   -49.420, E3 +318883.777}
SPL {X  -162.820, Y  +648.011, Z    +0.000, E1   -49.484, E3 +318895.454}
SPL {X  -162.820, Y  +655.976, Z    +0.000, E1   -49.445, E3 +318910.083}
SPL {X  -162.820, Y  +663.916, Z    +0.000, E1   -49.371, E3 +318924.512}
SPL {X  -162.820, Y  +669.755, Z    +0.000, E1   -49.387, E3 +318934.837}
SPL {X  -162.807, Y  +675.597, Z    +0.000, E1   -49.472, E3 +318944.739}
SPL {X  -162.632, Y  +681.322, Z    +0.000, E1   -49.345, E3 +318955.750}
SPL {X  -162.228, Y  +687.372, Z    +0.000, E1   -49.294, E3 +318966.837}
SPL {X  -161.723, Y  +692.372, Z    +0.000, E1   -49.172, E3 +318976.467}
SPL {X  -161.009, Y  +697.714, Z    +0.000, E1   -49.214, E3 +318985.752}
SPL {X  -160.313, Y  +701.965, Z    +0.000, E1   -48.932, E3 +318994.964}
SPL {X  -158.980, Y  +708.651, Z    +0.000, E1   -48.774, E3 +319008.004}
SPL {X  -157.477, Y  +714.869, Z    +0.000, E1   -48.424, E3 +319020.879}
SPL {X  -156.071, Y  +719.891, Z    +0.000, E1   -48.264, E3 +319030.755}
SPL {X  -154.661, Y  +724.395, Z    +0.000, E1   -47.951, E3 +319040.436}
SPL {X  -153.094, Y  +728.931, Z    +0.000, E1   -47.705, E3 +319049.873}
SPL {X  -151.300, Y  +733.655, Z    +0.000, E1   -47.339, E3 +319060.182}
SPL {X  -145.669, Y  +746.239, Z    +0.000, E1   -50.198, E3 +319066.958}
SPL {X  -135.084, Y  +764.399, Z    +0.000, E1   -44.787, E3 +319149.862}
ENDSPLINE

SPLINE
SPL {X  -153.038, Y  +729.086, Z    +0.000, E1   -30.522, E3 +319220.569}
SPL {X  -160.383, Y  +701.564, Z    +0.000, E1   -18.145, E3 +319230.605}
SPL {X  -162.078, Y  +689.023, Z    +0.000, E1   -11.510, E3 +319230.143}
SPL {X  -162.685, Y  +680.136, Z    +0.000, E1    -6.379, E3 +319230.432}
SPL {X  -162.820, Y  +672.919, Z    +0.000, E1    -1.752, E3 +319230.471}
SPL {X  -162.820, Y  +667.861, Z    +0.000, E1    +2.254, E3 +319230.272}
SPL {X  -162.820, Y  +662.755, Z    +0.000, E1    +7.521, E3 +319230.312}
SPL {X  -162.820, Y  +657.537, Z    +0.000, E1   +13.540, E3 +319229.982}
SPL {X  -162.820, Y  +650.460, Z    +0.000, E1   +22.200, E3 +319229.413}
SPL {X  -162.820, Y  +637.843, Z    +0.000, E1   +35.051, E3 +319231.490}
SPL {X  -162.820, Y  +595.072, Z    +0.000, E1   +53.652, E3 +319252.210}
SPL {X  -162.820, Y  +560.706, Z    +0.000, E1   +50.482, E3 +319313.119}
ENDSPLINE

SPLINE
SPL {X  -162.820, Y  +560.978, Z    +0.000, E1   +48.448, E3 +319325.204}
ENDSPLINE

SPLINE
SPL {X  -162.820, Y  +552.125, Z    +0.000, E1   +48.477, E3 +319341.309}
SPL {X  -162.820, Y  +545.800, Z    +0.000, E1   +48.334, E3 +319353.751}
SPL {X  -162.820, Y  +540.645, Z    +0.000, E1   +48.364, E3 +319363.102}
SPL {X  -162.820, Y  +534.689, Z    +0.000, E1   +48.295, E3 +319374.650}
SPL {X  -162.820, Y  +526.053, Z    +0.000, E1   +48.382, E3 +319390.225}
SPL {X  -162.820, Y  +519.666, Z    +0.000, E1   +48.261, E3 +319402.594}
SPL {X  -162.820, Y  +513.750, Z    +0.000, E1   +48.520, E3 +319412.037}
SPL {X  -162.820, Y  +508.282, Z    +0.000, E1   +48.307, E3 +319423.439}
SPL {X  -162.820, Y  +502.890, Z    +0.000, E1   +48.309, E3 +319433.366}
ENDSPLINE

SPLINE
SPL {X  -162.820, Y  +520.386, Z    +0.000, E1   +40.911, E3 +319440.095}
ENDSPLINE

SPLINE
SPL {X  -162.820, Y  +515.876, Z    +0.000, E1   +41.348, E3 +319448.294}
SPL {X  -162.820, Y  +507.007, Z    +0.000, E1   +42.470, E3 +319462.308}
SPL {X  -162.820, Y  +496.780, Z    +0.000, E1   +43.573, E3 +319478.563}
SPL {X  -162.820, Y  +488.962, Z    +0.000, E1   +44.342, E3 +319490.830}
SPL {X  -162.820, Y  +481.373, Z    +0.000, E1   +45.107, E3 +319502.315}
SPL {X  -162.820, Y  +473.909, Z    +0.000, E1   +45.743, E3 +319513.827}
SPL {X  -162.820, Y  +463.464, Z    +0.000, E1   +47.025, E3 +319527.044}
SPL {X  -162.820, Y  +451.336, Z    +0.000, E1   +48.248, E3 +319542.815}
SPL {X  -162.820, Y  +443.046, Z    +0.000, E1   +49.021, E3 +319553.314}
SPL {X  -162.820, Y  +435.978, Z    +0.000, E1   +49.560, E3 +319562.835}
SPL {X  -162.820, Y  +428.488, Z    +0.000, E1   +49.830, E3 +319574.414}
SPL {X  -162.820, Y  +423.062, Z    +0.000, E1   +49.728, E3 +319584.557}
SPL {X  -162.820, Y  +416.560, Z    +0.000, E1   +49.816, E3 +319595.538}
SPL {X  -162.820, Y  +407.996, Z    +0.000, E1   +49.793, E3 +319610.904}
SPL {X  -162.820, Y  +400.367, Z    +0.000, E1   +49.822, E3 +319623.962}
SPL {X  -162.820, Y  +393.582, Z    +0.000, E1   +49.779, E3 +319636.280}
SPL {X  -162.820, Y  +384.205, Z    +0.000, E1   +49.756, E3 +319653.061}
SPL {X  -162.753, Y  +375.844, Z    +0.000, E1   +49.816, E3 +319667.236}
SPL {X  -162.415, Y  +369.029, Z    +0.000, E1   +49.751, E3 +319679.725}
SPL {X  -161.760, Y  +361.947, Z    +0.000, E1   +49.515, E3 +319693.564}
SPL {X  -160.828, Y  +355.106, Z    +0.000, E1   +49.536, E3 +319705.480}
SPL {X  -159.832, Y  +349.452, Z    +0.000, E1   +49.188, E3 +319717.452}
SPL {X  -158.863, Y  +344.823, Z    +0.000, E1   +49.020, E3 +319726.501}
SPL {X  -157.695, Y  +339.971, Z    +0.000, E1   +48.934, E3 +319735.597}
SPL {X  -156.136, Y  +334.326, Z    +0.000, E1   +48.578, E3 +319747.563}
SPL {X  -154.561, Y  +329.302, Z    +0.000, E1   +48.290, E3 +319757.894}
SPL {X  -152.787, Y  +324.229, Z    +0.000, E1   +47.981, E3 +319768.584}
SPL {X  -150.789, Y  +319.074, Z    +0.000, E1   +47.585, E3 +319779.607}
SPL {X  -145.123, Y  +306.679, Z    +0.000, E1   +50.518, E3 +319785.504}
SPL {X  -135.207, Y  +289.783, Z    +0.000, E1   +44.101, E3 +319879.018}
ENDSPLINE

SPLINE
SPL {X  -154.528, Y  +329.203, Z    +0.000, E1   +28.834, E3 +319949.380}
SPL {X  -160.380, Y  +352.419, Z    +0.000, E1   +18.163, E3 +319953.740}
SPL {X  -162.408, Y  +368.921, Z    +0.000, E1    +9.337, E3 +319952.490}
SPL {X  -162.817, Y  +379.558, Z    +0.000, E1    +2.744, E3 +319952.880}
SPL {X  -162.820, Y  +384.383, Z    +0.000, E1    -0.869, E3 +319952.850}
SPL {X  -162.820, Y  +388.871, Z    +0.000, E1    -5.151, E3 +319952.556}
SPL {X  -162.820, Y  +395.861, Z    +0.000, E1   -13.028, E3 +319952.667}
SPL {X  -162.820, Y  +409.049, Z    +0.000, E1   -29.128, E3 +319951.510}
SPL {X  -162.820, Y  +444.592, Z    +0.000, E1   -49.032, E3 +319970.519}
SPL {X  -162.820, Y  +458.217, Z    +0.000, E1   -51.268, E3 +319982.465}
SPL {X  -162.820, Y  +501.848, Z    +0.000, E1   -54.235, E3 +320028.832}
ENDSPLINE

SPLINE
SPL {X  -162.820, Y  +498.156, Z    +0.000, E1   -50.986, E3 +320042.382}
ENDSPLINE

SPLINE
SPL {X  -162.820, Y  +499.429, Z    +0.000, E1   -49.453, E3 +320053.740}
SPL {X  -162.820, Y  +505.173, Z    +0.000, E1   -49.386, E3 +320064.396}
SPL {X  -162.820, Y  +510.642, Z    +0.000, E1   -49.447, E3 +320073.746}
SPL {X  -162.820, Y  +516.435, Z    +0.000, E1   -49.526, E3 +320083.624}
SPL {X  -162.820, Y  +523.383, Z    +0.000, E1   -49.407, E3 +320096.811}
SPL {X  -162.820, Y  +532.283, Z    +0.000, E1   -49.462, E3 +320112.413}
SPL {X  -162.820, Y  +541.471, Z    +0.000, E1   -49.456, E3 +320128.791}
SPL {X  -162.820, Y  +548.933, Z    +0.000, E1   -49.456, E3 +320141.980}
SPL {X  -162.820, Y  +553.997, Z    +0.000, E1   -49.325, E3 +320151.783}
SPL {X  -162.820, Y  +562.346, Z    +0.000, E1   -49.498, E3 +320165.846}
SPL {X  -162.820, Y  +570.444, Z    +0.000, E1   -49.421, E3 +320180.593}
SPL {X  -162.820, Y  +577.429, Z    +0.000, E1   -49.474, E3 +320192.707}
SPL {X  -162.820, Y  +585.965, Z    +0.000, E1   -49.447, E3 +320208.281}
SPL {X  -162.820, Y  +594.192, Z    +0.000, E1   -49.325, E3 +320223.524}
SPL {X  -162.820, Y  +600.267, Z    +0.000, E1   -49.443, E3 +320233.612}
SPL {X  -162.820, Y  +606.218, Z    +0.000, E1   -49.464, E3 +320244.159}
SPL {X  -162.820, Y  +612.538, Z    +0.000, E1   -49.488, E3 +320255.210}
SPL {X  -162.820, Y  +617.738, Z    +0.000, E1   -49.301, E3 +320265.647}
SPL {X  -162.820, Y  +624.265, Z    +0.000, E1   -49.443, E3 +320276.442}
SPL {X  -162.820, Y  +632.551, Z    +0.000, E1   -49.478, E3 +320291.211}
SPL {X  -162.820, Y  +641.207, Z    +0.000, E1   -49.420, E3 +320306.854}
SPL {X  -162.820, Y  +648.011, Z    +0.000, E1   -49.484, E3 +320318.531}
SPL {X  -162.820, Y  +655.976, Z    +0.000, E1   -49.445, E3 +320333.160}
SPL {X  -162.820, Y  +663.916, Z    +0.000, E1   -49.371, E3 +320347.589}
SPL {X  -162.820, Y  +669.755, Z    +0.000, E1   -49.387, E3 +320357.913}
SPL {X  -162.807, Y  +675.597, Z    +0.000, E1   -49.472, E3 +320367.816}
SPL {X  -162.632, Y  +681.322, Z    +0.000, E1   -49.345, E3 +320378.827}
SPL {X  -162.228, Y  +687.372, Z    +0.000, E1   -49.294, E3 +320389.914}
SPL {X  -161.723, Y  +692.372, Z    +0.000, E1   -49.172, E3 +320399.544}
SPL {X  -161.009, Y  +697.714, Z    +0.000, E1   -49.214, E3 +320408.828}
SPL {X  -160.313, Y  +701.965, Z    +0.000, E1   -48.932, E3 +320418.041}
SPL {X  -159.435, Y  +706.528, Z    +0.000, E1   -48.764, E3 +320427.167}
SPL {X  -157.894, Y  +713.249, Z    +0.000, E1   -48.586, E3 +320440.361}
SPL {X  -156.071, Y  +719.891, Z    +0.000, E1   -48.264, E3 +320453.832}
SPL {X  -154.661, Y  +724.395, Z    +0.000, E1   -47.951, E3 +320463.513}
SPL {X  -153.094, Y  +728.931, Z    +0.000, E1   -47.705, E3 +320472.950}
SPL {X  -151.300, Y  +733.655, Z    +0.000, E1   -47.339, E3 +320483.259}
SPL {X  -145.669, Y  +746.239, Z    +0.000, E1   -50.198, E3 +320490.035}
SPL {X  -135.559, Y  +763.690, Z    +0.000, E1   -44.340, E3 +320576.829}
ENDSPLINE

SPLINE
SPL {X  -153.801, Y  +726.938, Z    +0.000, E1   -29.643, E3 +320645.542}
SPL {X  -160.383, Y  +701.564, Z    +0.000, E1   -18.145, E3 +320653.682}
SPL {X  -162.078, Y  +689.023, Z    +0.000, E1   -11.510, E3 +320653.220}
SPL {X  -162.685, Y  +680.136, Z    +0.000, E1    -6.379, E3 +320653.509}
SPL {X  -162.820, Y  +672.919, Z    +0.000, E1    -1.752, E3 +320653.548}
SPL {X  -162.820, Y  +667.861, Z    +0.000, E1    +2.254, E3 +320653.349}
SPL {X  -162.820, Y  +662.755, Z    +0.000, E1    +7.521, E3 +320653.389}
SPL {X  -162.820, Y  +657.537, Z    +0.000, E1   +13.540, E3 +320653.059}
SPL {X  -162.820, Y  +650.460, Z    +0.000, E1   +22.200, E3 +320652.490}
SPL {X  -162.820, Y  +637.843, Z    +0.000, E1   +35.051, E3 +320654.566}
SPL {X  -162.820, Y  +595.072, Z    +0.000, E1   +53.652, E3 +320675.287}
SPL {X  -162.820, Y  +560.706, Z    +0.000, E1   +50.482, E3 +320736.196}
ENDSPLINE

SPLINE
SPL {X  -162.820, Y  +560.978, Z    +0.000, E1   +48.448, E3 +320748.281}
ENDSPLINE

SPLINE
SPL {X  -162.820, Y  +552.125, Z    +0.000, E1   +48.477, E3 +320764.386}
SPL {X  -162.820, Y  +545.800, Z    +0.000, E1   +48.334, E3 +320776.828}
SPL {X  -162.820, Y  +538.900, Z    +0.000, E1   +48.334, E3 +320789.743}
SPL {X  -162.820, Y  +530.572, Z    +0.000, E1   +48.392, E3 +320804.793}
SPL {X  -162.820, Y  +522.157, Z    +0.000, E1   +48.326, E3 +320820.882}
SPL {X  -162.820, Y  +512.600, Z    +0.000, E1   +48.469, E3 +320837.658}
SPL {X  -162.820, Y  +504.728, Z    +0.000, E1   +48.342, E3 +320852.987}
ENDSPLINE

SPLINE
SPL {X  -162.820, Y  +517.326, Z    +0.000, E1   +41.232, E3 +320868.707}
ENDSPLINE

SPLINE
SPL {X  -162.820, Y  +509.871, Z    +0.000, E1   +42.115, E3 +320880.808}
SPL {X  -162.820, Y  +501.934, Z    +0.000, E1   +43.022, E3 +320893.535}
SPL {X  -162.820, Y  +494.356, Z    +0.000, E1   +43.819, E3 +320905.376}
SPL {X  -162.820, Y  +487.058, Z    +0.000, E1   +44.544, E3 +320916.840}
SPL {X  -162.820, Y  +476.193, Z    +0.000, E1   +45.591, E3 +320933.279}
SPL {X  -162.820, Y  +465.836, Z    +0.000, E1   +46.727, E3 +320947.195}
SPL {X  -162.820, Y  +457.217, Z    +0.000, E1   +47.671, E3 +320958.233}
SPL {X  -162.820, Y  +446.677, Z    +0.000, E1   +48.707, E3 +320971.762}
SPL {X  -162.820, Y  +435.978, Z    +0.000, E1   +49.560, E3 +320985.912}
SPL {X  -162.820, Y  +428.488, Z    +0.000, E1   +49.830, E3 +320997.491}
SPL {X  -162.820, Y  +423.062, Z    +0.000, E1   +49.728, E3 +321007.634}
SPL {X  -162.820, Y  +416.560, Z    +0.000, E1   +49.816, E3 +321018.615}
SPL {X  -162.820, Y  +407.996, Z    +0.000, E1   +49.793, E3 +321033.981}
SPL {X  -162.820, Y  +398.766, Z    +0.000, E1   +49.793, E3 +321050.160}
SPL {X  -162.820, Y  +391.831, Z    +0.000, E1   +49.801, E3 +321062.206}
SPL {X  -162.820, Y  +386.334, Z    +0.000, E1   +49.739, E3 +321072.294}
SPL {X  -162.801, Y  +377.981, Z    +0.000, E1   +49.798, E3 +321086.816}
SPL {X  -162.314, Y  +367.677, Z    +0.000, E1   +49.734, E3 +321105.456}
SPL {X  -161.359, Y  +358.734, Z    +0.000, E1   +49.535, E3 +321122.239}
SPL {X  -160.051, Y  +350.597, Z    +0.000, E1   +49.332, E3 +321137.850}
SPL {X  -158.863, Y  +344.823, Z    +0.000, E1   +49.020, E3 +321149.578}
SPL {X  -157.695, Y  +339.971, Z    +0.000, E1   +48.934, E3 +321158.674}
SPL {X  -156.496, Y  +335.563, Z    +0.000, E1   +48.599, E3 +321168.251}
SPL {X  -154.894, Y  +330.318, Z    +0.000, E1   +48.380, E3 +321178.794}
SPL {X  -153.352, Y  +325.786, Z    +0.000, E1   +48.028, E3 +321188.551}
SPL {X  -151.316, Y  +320.384, Z    +0.000, E1   +47.734, E3 +321199.766}
SPL {X  -145.123, Y  +306.679, Z    +0.000, E1   +50.518, E3 +321208.581}
SPL {X  -135.207, Y  +289.783, Z    +0.000, E1   +44.101, E3 +321302.095}
ENDSPLINE

SPLINE
SPL {X  -154.528, Y  +329.203, Z    +0.000, E1   +28.834, E3 +321372.456}
SPL {X  -160.380, Y  +352.419, Z    +0.000, E1   +18.163, E3 +321376.817}
SPL {X  -162.149, Y  +365.734, Z    +0.000, E1   +11.090, E3 +321375.425}
SPL {X  -162.754, Y  +375.862, Z    +0.000, E1    +5.134, E3 +321376.262}
SPL {X  -162.820, Y  +382.085, Z    +0.000, E1    +0.928, E3 +321375.951}
SPL {X  -162.820, Y  +385.149, Z    +0.000, E1    -1.602, E3 +321375.678}
SPL {X  -162.820, Y  +388.871, Z    +0.000, E1    -5.151, E3 +321375.633}
SPL {X  -162.820, Y  +395.861, Z    +0.000, E1   -13.028, E3 +321375.744}
SPL {X  -162.820, Y  +409.049, Z    +0.000, E1   -29.128, E3 +321374.587}
SPL {X  -162.820, Y  +446.299, Z    +0.000, E1   -49.360, E3 +321395.090}
SPL {X  -162.820, Y  +502.427, Z    +0.000, E1   -53.345, E3 +321458.075}
ENDSPLINE

SPLINE
SPL {X  -162.820, Y  +494.458, Z    +0.000, E1   -49.332, E3 +321468.608}
ENDSPLINE

SPLINE
SPL {X  -162.820, Y  +499.429, Z    +0.000, E1   -49.453, E3 +321476.817}
SPL {X  -162.820, Y  +505.173, Z    +0.000, E1   -49.386, E3 +321487.473}
SPL {X  -162.820, Y  +510.642, Z    +0.000, E1   -49.447, E3 +321496.823}
SPL {X  -162.820, Y  +516.435, Z    +0.000, E1   -49.526, E3 +321506.701}
SPL {X  -162.820, Y  +523.383, Z    +0.000, E1   -49.407, E3 +321519.888}
SPL {X  -162.820, Y  +530.598, Z    +0.000, E1   -49.471, E3 +321532.289}
SPL {X  -162.820, Y  +536.932, Z    +0.000, E1   -49.395, E3 +321544.047}
SPL {X  -162.820, Y  +543.021, Z    +0.000, E1   -49.432, E3 +321554.653}
SPL {X  -162.820, Y  +548.933, Z    +0.000, E1   -49.456, E3 +321565.057}
SPL {X  -162.820, Y  +553.997, Z    +0.000, E1   -49.325, E3 +321574.860}
SPL {X  -162.820, Y  +560.268, Z    +0.000, E1   -49.531, E3 +321584.818}
SPL {X  -162.820, Y  +564.590, Z    +0.000, E1   -49.361, E3 +321593.518}
SPL {X  -162.820, Y  +570.444, Z    +0.000, E1   -49.421, E3 +321603.670}
SPL {X  -162.820, Y  +577.429, Z    +0.000, E1   -49.474, E3 +321615.784}
SPL {X  -162.820, Y  +585.965, Z    +0.000, E1   -49.447, E3 +321631.358}
SPL {X  -162.820, Y  +594.192, Z    +0.000, E1   -49.325, E3 +321646.601}
SPL {X  -162.820, Y  +600.267, Z    +0.000, E1   -49.443, E3 +321656.689}
SPL {X  -162.820, Y  +606.218, Z    +0.000, E1   -49.464, E3 +321667.236}
SPL {X  -162.820, Y  +612.538, Z    +0.000, E1   -49.488, E3 +321678.287}
SPL {X  -162.820, Y  +617.738, Z    +0.000, E1   -49.301, E3 +321688.723}
SPL {X  -162.820, Y  +624.265, Z    +0.000, E1   -49.443, E3 +321699.519}
SPL {X  -162.820, Y  +632.551, Z    +0.000, E1   -49.478, E3 +321714.288}
SPL {X  -162.820, Y  +641.207, Z    +0.000, E1   -49.420, E3 +321729.931}
SPL {X  -162.820, Y  +649.864, Z    +0.000, E1   -49.433, E3 +321745.409}
SPL {X  -162.820, Y  +658.147, Z    +0.000, E1   -49.491, E3 +321759.676}
SPL {X  -162.820, Y  +663.916, Z    +0.000, E1   -49.371, E3 +321770.666}
SPL {X  -162.820, Y  +669.755, Z    +0.000, E1   -49.387, E3 +321780.990}
SPL {X  -162.807, Y  +675.597, Z    +0.000, E1   -49.472, E3 +321790.893}
SPL {X  -162.632, Y  +681.322, Z    +0.000, E1   -49.345, E3 +321801.904}
SPL {X  -162.228, Y  +687.372, Z    +0.000, E1   -49.294, E3 +321812.991}
SPL {X  -161.723, Y  +692.372, Z    +0.000, E1   -49.172, E3 +321822.621}
SPL {X  -161.009, Y  +697.714, Z    +0.000, E1   -49.214, E3 +321831.905}
SPL {X  -160.313, Y  +701.965, Z    +0.000, E1   -48.932, E3 +321841.118}
SPL {X  -158.980, Y  +708.651, Z    +0.000, E1   -48.774, E3 +321854.158}
SPL {X  -157.477, Y  +714.869, Z    +0.000, E1   -48.424, E3 +321867.032}
SPL {X  -156.071, Y  +719.891, Z    +0.000, E1   -48.264, E3 +321876.909}
SPL {X  -154.661, Y  +724.395, Z    +0.000, E1   -47.951, E3 +321886.590}
SPL {X  -153.094, Y  +728.931, Z    +0.000, E1   -47.705, E3 +321896.027}
SPL {X  -150.266, Y  +736.194, Z    +0.000, E1   -47.943, E3 +321907.636}
SPL {X  -143.458, Y  +750.508, Z    +0.000, E1   -51.034, E3 +321915.661}
SPL {X  -135.559, Y  +763.690, Z    +0.000, E1   -44.340, E3 +321999.906}
ENDSPLINE

SPLINE
SPL {X  -153.801, Y  +726.938, Z    +0.000, E1   -29.643, E3 +322068.619}
SPL {X  -160.383, Y  +701.564, Z    +0.000, E1   -18.145, E3 +322076.759}
SPL {X  -162.078, Y  +689.023, Z    +0.000, E1   -11.510, E3 +322076.297}
SPL {X  -162.685, Y  +680.136, Z    +0.000, E1    -6.379, E3 +322076.585}
SPL {X  -162.820, Y  +672.919, Z    +0.000, E1    -1.752, E3 +322076.624}
SPL {X  -162.820, Y  +667.861, Z    +0.000, E1    +2.254, E3 +322076.426}
SPL {X  -162.820, Y  +662.755, Z    +0.000, E1    +7.521, E3 +322076.466}
SPL {X  -162.820, Y  +657.537, Z    +0.000, E1   +13.540, E3 +322076.136}
SPL {X  -162.820, Y  +650.460, Z    +0.000, E1   +22.200, E3 +322075.567}
SPL {X  -162.820, Y  +637.843, Z    +0.000, E1   +35.051, E3 +322077.643}
SPL {X  -162.820, Y  +595.072, Z    +0.000, E1   +53.652, E3 +322098.364}
SPL {X  -162.820, Y  +561.831, Z    +0.000, E1   +49.171, E3 +322165.586}
SPL {X  -162.820, Y  +553.813, Z    +0.000, E1   +48.452, E3 +322184.651}
SPL {X  -162.820, Y  +543.226, Z    +0.000, E1   +48.398, E3 +322204.503}
SPL {X  -162.820, Y  +534.689, Z    +0.000, E1   +48.295, E3 +322220.804}
SPL {X  -162.820, Y  +528.564, Z    +0.000, E1   +48.407, E3 +322231.378}
SPL {X  -162.820, Y  +522.157, Z    +0.000, E1   +48.326, E3 +322243.959}
SPL {X  -162.820, Y  +513.750, Z    +0.000, E1   +48.520, E3 +322258.191}
SPL {X  -162.820, Y  +508.282, Z    +0.000, E1   +48.307, E3 +322269.593}
SPL {X  -162.820, Y  +502.890, Z    +0.000, E1   +48.309, E3 +322279.519}
ENDSPLINE

SPLINE
SPL {X  -162.820, Y  +520.386, Z    +0.000, E1   +40.911, E3 +322286.249}
ENDSPLINE

SPLINE
SPL {X  -162.820, Y  +515.876, Z    +0.000, E1   +41.348, E3 +322294.447}
SPL {X  -162.820, Y  +507.007, Z    +0.000, E1   +42.470, E3 +322308.462}
SPL {X  -162.820, Y  +496.780, Z    +0.000, E1   +43.573, E3 +322324.717}
SPL {X  -162.820, Y  +488.962, Z    +0.000, E1   +44.342, E3 +322336.984}
SPL {X  -162.820, Y  +481.373, Z    +0.000, E1   +45.107, E3 +322348.469}
SPL {X  -162.820, Y  +473.909, Z    +0.000, E1   +45.743, E3 +322359.981}
SPL {X  -162.820, Y  +465.836, Z    +0.000, E1   +46.727, E3 +322370.272}
SPL {X  -162.820, Y  +457.217, Z    +0.000, E1   +47.671, E3 +322381.310}
SPL {X  -162.820, Y  +449.104, Z    +0.000, E1   +48.459, E3 +322391.779}
SPL {X  -162.820, Y  +438.072, Z    +0.000, E1   +49.432, E3 +322406.133}
SPL {X  -162.820, Y  +428.488, Z    +0.000, E1   +49.830, E3 +322420.568}
SPL {X  -162.820, Y  +423.062, Z    +0.000, E1   +49.728, E3 +322430.711}
SPL {X  -162.820, Y  +416.560, Z    +0.000, E1   +49.816, E3 +322441.692}
SPL {X  -162.820, Y  +410.559, Z    +0.000, E1   +49.727, E3 +322452.748}
SPL {X  -162.820, Y  +405.170, Z    +0.000, E1   +49.772, E3 +322461.949}
SPL {X  -162.820, Y  +398.766, Z    +0.000, E1   +49.793, E3 +322473.237}
SPL {X  -162.820, Y  +391.831, Z    +0.000, E1   +49.801, E3 +322485.283}
SPL {X  -162.820, Y  +386.334, Z    +0.000, E1   +49.739, E3 +322495.371}
SPL {X  -162.801, Y  +377.981, Z    +0.000, E1   +49.798, E3 +322509.893}
SPL {X  -162.314, Y  +367.677, Z    +0.000, E1   +49.734, E3 +322528.533}
SPL {X  -161.614, Y  +360.718, Z    +0.000, E1   +49.491, E3 +322541.950}
SPL {X  -160.828, Y  +355.106, Z    +0.000, E1   +49.536, E3 +322551.634}
SPL {X  -159.832, Y  +349.452, Z    +0.000, E1   +49.188, E3 +322563.606}
SPL {X  -158.863, Y  +344.823, Z    +0.000, E1   +49.020, E3 +322572.655}
SPL {X  -157.695, Y  +339.971, Z    +0.000, E1   +48.934, E3 +322581.751}
SPL {X  -156.136, Y  +334.326, Z    +0.000, E1   +48.578, E3 +322593.717}
SPL {X  -154.561, Y  +329.302, Z    +0.000, E1   +48.290, E3 +322604.048}
SPL {X  -152.787, Y  +324.229, Z    +0.000, E1   +47.981, E3 +322614.738}
SPL {X  -150.789, Y  +319.074, Z    +0.000, E1   +47.585, E3 +322625.760}
SPL {X  -145.123, Y  +306.679, Z    +0.000, E1   +50.518, E3 +322631.658}
SPL {X  -135.207, Y  +289.783, Z    +0.000, E1   +44.101, E3 +322725.172}
ENDSPLINE

SPLINE
SPL {X  -154.528, Y  +329.203, Z    +0.000, E1   +28.834, E3 +322795.533}
SPL {X  -160.380, Y  +352.419, Z    +0.000, E1   +18.163, E3 +322799.894}
SPL {X  -162.408, Y  +368.921, Z    +0.000, E1    +9.337, E3 +322798.644}
SPL {X  -162.817, Y  +379.558, Z    +0.000, E1    +2.744, E3 +322799.034}
SPL {X  -162.820, Y  +383.077, Z    +0.000, E1    +0.110, E3 +322799.429}
SPL {X  -162.820, Y  +386.028, Z    +0.000, E1    -2.328, E3 +322798.752}
SPL {X  -162.820, Y  +389.792, Z    +0.000, E1    -6.211, E3 +322798.684}
SPL {X  -162.820, Y  +394.068, Z    +0.000, E1   -11.043, E3 +322798.801}
SPL {X  -162.820, Y  +398.921, Z    +0.000, E1   -16.945, E3 +322798.854}
SPL {X  -162.820, Y  +409.049, Z    +0.000, E1   -29.128, E3 +322797.663}
SPL {X  -162.820, Y  +444.592, Z    +0.000, E1   -49.032, E3 +322816.673}
SPL {X  -162.820, Y  +458.217, Z    +0.000, E1   -51.268, E3 +322828.618}
SPL {X  -162.820, Y  +501.848, Z    +0.000, E1   -54.235, E3 +322874.986}
ENDSPLINE

SPLINE
SPL {X  -162.820, Y  +498.156, Z    +0.000, E1   -50.986, E3 +322888.536}
ENDSPLINE

SPLINE
SPL {X  -162.820, Y  +499.429, Z    +0.000, E1   -49.453, E3 +322899.894}
SPL {X  -162.820, Y  +505.173, Z    +0.000, E1   -49.386, E3 +322910.550}
SPL {X  -162.820, Y  +510.642, Z    +0.000, E1   -49.447, E3 +322919.900}
SPL {X  -162.820, Y  +516.435, Z    +0.000, E1   -49.526, E3 +322929.778}
SPL {X  -162.820, Y  +523.383, Z    +0.000, E1   -49.407, E3 +322942.965}
SPL {X  -162.820, Y  +532.283, Z    +0.000, E1   -49.462, E3 +322958.567}
SPL {X  -162.820, Y  +541.471, Z    +0.000, E1   -49.456, E3 +322974.945}
SPL {X  -162.820, Y  +548.933, Z    +0.000, E1   -49.456, E3 +322988.134}
SPL {X  -162.820, Y  +553.997, Z    +0.000, E1   -49.325, E3 +322997.937}
SPL {X  -162.820, Y  +562.346, Z    +0.000, E1   -49.498, E3 +323012.000}
SPL {X  -162.820, Y  +570.444, Z    +0.000, E1   -49.421, E3 +323026.747}
SPL {X  -162.820, Y  +577.429, Z    +0.000, E1   -49.474, E3 +323038.861}
SPL {X  -162.820, Y  +585.965, Z    +0.000, E1   -49.447, E3 +323054.435}
SPL {X  -162.820, Y  +594.192, Z    +0.000, E1   -49.325, E3 +323069.678}
SPL {X  -162.820, Y  +600.267, Z    +0.000, E1   -49.443, E3 +323079.766}
SPL {X  -162.820, Y  +606.218, Z    +0.000, E1   -49.464, E3 +323090.313}
SPL {X  -162.820, Y  +612.538, Z    +0.000, E1   -49.488, E3 +323101.364}
SPL {X  -162.820, Y  +617.738, Z    +0.000, E1   -49.301, E3 +323111.800}
SPL {X  -162.820, Y  +624.265, Z    +0.000, E1   -49.443, E3 +323122.596}
SPL {X  -162.820, Y  +632.551, Z    +0.000, E1   -49.478, E3 +323137.364}
SPL {X  -162.820, Y  +641.207, Z    +0.000, E1   -49.420, E3 +323153.008}
SPL {X  -162.820, Y  +648.011, Z    +0.000, E1   -49.484, E3 +323164.685}
SPL {X  -162.820, Y  +655.976, Z    +0.000, E1   -49.445, E3 +323179.314}
SPL {X  -162.820, Y  +663.916, Z    +0.000, E1   -49.371, E3 +323193.743}
SPL {X  -162.820, Y  +669.755, Z    +0.000, E1   -49.387, E3 +323204.067}
SPL {X  -162.807, Y  +675.597, Z    +0.000, E1   -49.472, E3 +323213.970}
SPL {X  -162.632, Y  +681.322, Z    +0.000, E1   -49.345, E3 +323224.981}
SPL {X  -162.228, Y  +687.372, Z    +0.000, E1   -49.294, E3 +323236.068}
SPL {X  -161.723, Y  +692.372, Z    +0.000, E1   -49.172, E3 +323245.698}
SPL {X  -161.009, Y  +697.714, Z    +0.000, E1   -49.214, E3 +323254.982}
SPL {X  -160.313, Y  +701.965, Z    +0.000, E1   -48.932, E3 +323264.194}
SPL {X  -158.980, Y  +708.651, Z    +0.000, E1   -48.774, E3 +323277.235}
SPL {X  -157.477, Y  +714.869, Z    +0.000, E1   -48.424, E3 +323290.109}
SPL {X  -156.071, Y  +719.891, Z    +0.000, E1   -48.264, E3 +323299.986}
SPL {X  -154.661, Y  +724.395, Z    +0.000, E1   -47.951, E3 +323309.667}
SPL {X  -153.094, Y  +728.931, Z    +0.000, E1   -47.705, E3 +323319.104}
SPL {X  -150.266, Y  +736.194, Z    +0.000, E1   -47.943, E3 +323330.713}
SPL {X  -143.458, Y  +750.508, Z    +0.000, E1   -51.034, E3 +323338.738}
SPL {X  -135.084, Y  +764.399, Z    +0.000, E1   -44.787, E3 +323419.093}
ENDSPLINE

SPLINE
SPL {X  -153.038, Y  +729.086, Z    +0.000, E1   -30.522, E3 +323489.800}
SPL {X  -160.383, Y  +701.564, Z    +0.000, E1   -18.145, E3 +323499.836}
SPL {X  -162.078, Y  +689.023, Z    +0.000, E1   -11.510, E3 +323499.374}
SPL {X  -162.685, Y  +680.136, Z    +0.000, E1    -6.379, E3 +323499.662}
SPL {X  -162.820, Y  +672.919, Z    +0.000, E1    -1.752, E3 +323499.701}
SPL {X  -162.820, Y  +667.861, Z    +0.000, E1    +2.254, E3 +323499.503}
SPL {X  -162.820, Y  +662.755, Z    +0.000, E1    +7.521, E3 +323499.543}
SPL {X  -162.820, Y  +657.537, Z    +0.000, E1   +13.540, E3 +323499.212}
SPL {X  -162.820, Y  +650.460, Z    +0.000, E1   +22.200, E3 +323498.643}
SPL {X  -162.820, Y  +637.843, Z    +0.000, E1   +35.051, E3 +323500.720}
SPL {X  -162.820, Y  +595.072, Z    +0.000, E1   +53.652, E3 +323521.440}
SPL {X  -162.820, Y  +561.831, Z    +0.000, E1   +49.171, E3 +323588.663}
SPL {X  -162.820, Y  +553.813, Z    +0.000, E1   +48.452, E3 +323607.728}
SPL {X  -162.820, Y  +543.226, Z    +0.000, E1   +48.398, E3 +323627.580}
SPL {X  -162.820, Y  +534.689, Z    +0.000, E1   +48.295, E3 +323643.881}
SPL {X  -162.820, Y  +528.564, Z    +0.000, E1   +48.407, E3 +323654.455}
SPL {X  -162.820, Y  +522.157, Z    +0.000, E1   +48.326, E3 +323667.036}
SPL {X  -162.820, Y  +513.750, Z    +0.000, E1   +48.520, E3 +323681.268}
SPL {X  -162.820, Y  +508.282, Z    +0.000, E1   +48.307, E3 +323692.670}
SPL {X  -162.820, Y  +502.890, Z    +0.000, E1   +48.309, E3 +323702.596}
ENDSPLINE

SPLINE
SPL {X  -162.820, Y  +520.386, Z    +0.000, E1   +40.911, E3 +323709.326}
ENDSPLINE

SPLINE
SPL {X  -162.820, Y  +515.876, Z    +0.000, E1   +41.348, E3 +323717.524}
SPL {X  -162.820, Y  +507.007, Z    +0.000, E1   +42.470, E3 +323731.539}
SPL {X  -162.820, Y  +496.780, Z    +0.000, E1   +43.573, E3 +323747.793}
SPL {X  -162.820, Y  +488.962, Z    +0.000, E1   +44.342, E3 +323760.061}
SPL {X  -162.820, Y  +481.373, Z    +0.000, E1   +45.107, E3 +323771.545}
SPL {X  -162.820, Y  +473.909, Z    +0.000, E1   +45.743, E3 +323783.058}
SPL {X  -162.820, Y  +465.836, Z    +0.000, E1   +46.727, E3 +323793.349}
SPL {X  -162.820, Y  +457.217, Z    +0.000, E1   +47.671, E3 +323804.387}
SPL {X  -162.820, Y  +449.104, Z    +0.000, E1   +48.459, E3 +323814.855}
SPL {X  -162.820, Y  +438.072, Z    +0.000, E1   +49.432, E3 +323829.210}
SPL {X  -162.820, Y  +428.488, Z    +0.000, E1   +49.830, E3 +323843.645}
SPL {X  -162.820, Y  +423.062, Z    +0.000, E1   +49.728, E3 +323853.788}
SPL {X  -162.820, Y  +416.560, Z    +0.000, E1   +49.816, E3 +323864.769}
SPL {X  -162.820, Y  +410.559, Z    +0.000, E1   +49.727, E3 +323875.824}
SPL {X  -162.820, Y  +405.170, Z    +0.000, E1   +49.772, E3 +323885.026}
SPL {X  -162.820, Y  +398.766, Z    +0.000, E1   +49.793, E3 +323896.314}
SPL {X  -162.820, Y  +391.831, Z    +0.000, E1   +49.801, E3 +323908.360}
SPL {X  -162.820, Y  +386.334, Z    +0.000, E1   +49.739, E3 +323918.448}
SPL {X  -162.801, Y  +377.981, Z    +0.000, E1   +49.798, E3 +323932.970}
SPL {X  -162.314, Y  +367.677, Z    +0.000, E1   +49.734, E3 +323951.610}
SPL {X  -161.614, Y  +360.718, Z    +0.000, E1   +49.491, E3 +323965.027}
SPL {X  -160.828, Y  +355.106, Z    +0.000, E1   +49.536, E3 +323974.711}
SPL {X  -159.832, Y  +349.452, Z    +0.000, E1   +49.188, E3 +323986.682}
SPL {X  -158.863, Y  +344.823, Z    +0.000, E1   +49.020, E3 +323995.732}
SPL {X  -157.695, Y  +339.971, Z    +0.000, E1   +48.934, E3 +324004.828}
SPL {X  -156.496, Y  +335.563, Z    +0.000, E1   +48.599, E3 +324014.405}
SPL {X  -154.894, Y  +330.318, Z    +0.000, E1   +48.380, E3 +324024.948}
SPL {X  -153.352, Y  +325.786, Z    +0.000, E1   +48.028, E3 +324034.705}
SPL {X  -151.655, Y  +321.245, Z    +0.000, E1   +47.770, E3 +324044.126}
SPL {X  -148.347, Y  +313.391, Z    +0.000, E1   +48.924, E3 +324051.723}
SPL {X  -143.047, Y  +302.732, Z    +0.000, E1   +51.043, E3 +324058.243}
SPL {X  -135.207, Y  +289.783, Z    +0.000, E1   +44.101, E3 +324148.249}
ENDSPLINE

SPLINE
SPL {X  -154.528, Y  +329.203, Z    +0.000, E1   +28.834, E3 +324218.610}
SPL {X  -160.380, Y  +352.419, Z    +0.000, E1   +18.163, E3 +324222.971}
SPL {X  -162.408, Y  +368.921, Z    +0.000, E1    +9.337, E3 +324221.721}
SPL {X  -162.817, Y  +379.558, Z    +0.000, E1    +2.744, E3 +324222.111}
SPL {X  -162.820, Y  +383.077, Z    +0.000, E1    +0.110, E3 +324222.506}
SPL {X  -162.820, Y  +386.028, Z    +0.000, E1    -2.328, E3 +324221.829}
SPL {X  -162.820, Y  +389.792, Z    +0.000, E1    -6.211, E3 +324221.761}
SPL {X  -162.820, Y  +394.068, Z    +0.000, E1   -11.043, E3 +324221.878}
SPL {X  -162.820, Y  +398.921, Z    +0.000, E1   -16.945, E3 +324221.931}
SPL {X  -162.820, Y  +409.049, Z    +0.000, E1   -29.128, E3 +324220.740}
SPL {X  -162.820, Y  +446.299, Z    +0.000, E1   -49.360, E3 +324241.244}
SPL {X  -162.820, Y  +502.427, Z    +0.000, E1   -53.345, E3 +324304.229}
ENDSPLINE

SPLINE
SPL {X  -162.820, Y  +494.458, Z    +0.000, E1   -49.332, E3 +324314.761}
ENDSPLINE

SPLINE
SPL {X  -162.820, Y  +499.429, Z    +0.000, E1   -49.453, E3 +324322.971}
SPL {X  -162.820, Y  +507.703, Z    +0.000, E1   -49.462, E3 +324337.886}
SPL {X  -162.820, Y  +516.435, Z    +0.000, E1   -49.526, E3 +324352.855}
SPL {X  -162.820, Y  +522.095, Z    +0.000, E1   -49.420, E3 +324363.551}
SPL {X  -162.820, Y  +529.397, Z    +0.000, E1   -49.440, E3 +324376.560}
SPL {X  -162.820, Y  +535.099, Z    +0.000, E1   -49.339, E3 +324387.178}
SPL {X  -162.820, Y  +541.471, Z    +0.000, E1   -49.456, E3 +324398.022}
SPL {X  -162.820, Y  +548.933, Z    +0.000, E1   -49.456, E3 +324411.210}
SPL {X  -162.820, Y  +553.997, Z    +0.000, E1   -49.325, E3 +324421.014}
SPL {X  -162.820, Y  +562.346, Z    +0.000, E1   -49.498, E3 +324435.077}
SPL {X  -162.820, Y  +570.444, Z    +0.000, E1   -49.421, E3 +324449.823}
SPL {X  -162.820, Y  +577.429, Z    +0.000, E1   -49.474, E3 +324461.938}
SPL {X  -162.820, Y  +585.965, Z    +0.000, E1   -49.447, E3 +324477.512}
SPL {X  -162.820, Y  +594.192, Z    +0.000, E1   -49.325, E3 +324492.755}
SPL {X  -162.820, Y  +600.267, Z    +0.000, E1   -49.443, E3 +324502.843}
SPL {X  -162.820, Y  +606.218, Z    +0.000, E1   -49.464, E3 +324513.390}
SPL {X  -162.820, Y  +612.538, Z    +0.000, E1   -49.488, E3 +324524.441}
SPL {X  -162.820, Y  +617.738, Z    +0.000, E1   -49.301, E3 +324534.877}
SPL {X  -162.820, Y  +624.265, Z    +0.000, E1   -49.443, E3 +324545.673}
SPL {X  -162.820, Y  +632.551, Z    +0.000, E1   -49.478, E3 +324560.441}
SPL {X  -162.820, Y  +641.207, Z    +0.000, E1   -49.420, E3 +324576.085}
SPL {X  -162.820, Y  +648.011, Z    +0.000, E1   -49.484, E3 +324587.762}
SPL {X  -162.820, Y  +655.976, Z    +0.000, E1   -49.445, E3 +324602.390}
SPL {X  -162.820, Y  +663.916, Z    +0.000, E1   -49.371, E3 +324616.819}
SPL {X  -162.820, Y  +669.755, Z    +0.000, E1   -49.387, E3 +324627.144}
SPL {X  -162.807, Y  +675.597, Z    +0.000, E1   -49.472, E3 +324637.047}
SPL {X  -162.632, Y  +681.322, Z    +0.000, E1   -49.345, E3 +324648.058}
SPL {X  -162.228, Y  +687.372, Z    +0.000, E1   -49.294, E3 +324659.145}
SPL {X  -161.723, Y  +692.372, Z    +0.000, E1   -49.172, E3 +324668.775}
SPL {X  -161.009, Y  +697.714, Z    +0.000, E1   -49.214, E3 +324678.059}
SPL {X  -160.313, Y  +701.965, Z    +0.000, E1   -48.932, E3 +324687.271}
SPL {X  -158.980, Y  +708.651, Z    +0.000, E1   -48.774, E3 +324700.312}
SPL {X  -157.477, Y  +714.869, Z    +0.000, E1   -48.424, E3 +324713.186}
SPL {X  -156.071, Y  +719.891, Z    +0.000, E1   -48.264, E3 +324723.063}
SPL {X  -154.661, Y  +724.395, Z    +0.000, E1   -47.951, E3 +324732.744}
SPL {X  -153.094, Y  +728.931, Z    +0.000, E1   -47.705, E3 +324742.181}
SPL {X  -150.266, Y  +736.194, Z    +0.000, E1   -47.943, E3 +324753.789}
SPL {X  -143.458, Y  +750.508, Z    +0.000, E1   -51.034, E3 +324761.815}
SPL {X  -135.084, Y  +764.399, Z    +0.000, E1   -44.787, E3 +324842.170}
ENDSPLINE

SPLINE
SPL {X  -153.038, Y  +729.086, Z    +0.000, E1   -30.522, E3 +324912.877}
SPL {X  -160.383, Y  +701.564, Z    +0.000, E1   -18.145, E3 +324922.913}
SPL {X  -162.078, Y  +689.023, Z    +0.000, E1   -11.510, E3 +324922.451}
SPL {X  -162.685, Y  +680.136, Z    +0.000, E1    -6.379, E3 +324922.739}
SPL {X  -162.820, Y  +672.919, Z    +0.000, E1    -1.752, E3 +324922.778}
SPL {X  -162.820, Y  +667.861, Z    +0.000, E1    +2.254, E3 +324922.579}
SPL {X  -162.820, Y  +662.755, Z    +0.000, E1    +7.521, E3 +324922.620}
SPL {X  -162.820, Y  +657.537, Z    +0.000, E1   +13.540, E3 +324922.289}
SPL {X  -162.820, Y  +650.460, Z    +0.000, E1   +22.200, E3 +324921.720}
SPL {X  -162.820, Y  +637.843, Z    +0.000, E1   +35.051, E3 +324923.797}
SPL {X  -162.820, Y  +595.072, Z    +0.000, E1   +53.652, E3 +324944.517}
SPL {X  -162.820, Y  +561.831, Z    +0.000, E1   +49.171, E3 +325011.740}
SPL {X  -162.820, Y  +553.813, Z    +0.000, E1   +48.452, E3 +325030.805}
SPL {X  -162.820, Y  +543.226, Z    +0.000, E1   +48.398, E3 +325050.657}
SPL {X  -162.820, Y  +534.689, Z    +0.000, E1   +48.295, E3 +325066.958}
SPL {X  -162.820, Y  +528.564, Z    +0.000, E1   +48.407, E3 +325077.531}
SPL {X  -162.820, Y  +522.157, Z    +0.000, E1   +48.326, E3 +325090.113}
SPL {X  -162.820, Y  +513.750, Z    +0.000, E1   +48.520, E3 +325104.344}
SPL {X  -162.820, Y  +508.282, Z    +0.000, E1   +48.307, E3 +325115.747}
SPL {X  -162.820, Y  +502.890, Z    +0.000, E1   +48.309, E3 +325125.673}
ENDSPLINE

SPLINE
SPL {X  -162.820, Y  +520.386, Z    +0.000, E1   +40.911, E3 +325132.403}
ENDSPLINE

SPLINE
SPL {X  -162.820, Y  +515.876, Z    +0.000, E1   +41.348, E3 +325140.601}
SPL {X  -162.820, Y  +507.007, Z    +0.000, E1   +42.470, E3 +325154.615}
SPL {X  -162.820, Y  +496.780, Z    +0.000, E1   +43.573, E3 +325170.870}
SPL {X  -162.820, Y  +488.962, Z    +0.000, E1   +44.342, E3 +325183.138}
SPL {X  -162.820, Y  +481.373, Z    +0.000, E1   +45.107, E3 +325194.622}
SPL {X  -162.820, Y  +473.909, Z    +0.000, E1   +45.743, E3 +325206.135}
SPL {X  -162.820, Y  +465.836, Z    +0.000, E1   +46.727, E3 +325216.426}
SPL {X  -162.820, Y  +457.217, Z    +0.000, E1   +47.671, E3 +325227.464}
SPL {X  -162.820, Y  +449.104, Z    +0.000, E1   +48.459, E3 +325237.932}
SPL {X  -162.820, Y  +438.072, Z    +0.000, E1   +49.432, E3 +325252.287}
SPL {X  -162.820, Y  +428.488, Z    +0.000, E1   +49.830, E3 +325266.722}
SPL {X  -162.820, Y  +423.062, Z    +0.000, E1   +49.728, E3 +325276.865}
SPL {X  -162.820, Y  +416.560, Z    +0.000, E1   +49.816, E3 +325287.846}
SPL {X  -162.820, Y  +410.559, Z    +0.000, E1   +49.727, E3 +325298.901}
SPL {X  -162.820, Y  +405.170, Z    +0.000, E1   +49.772, E3 +325308.103}
SPL {X  -162.820, Y  +398.766, Z    +0.000, E1   +49.793, E3 +325319.391}
SPL {X  -162.820, Y  +391.831, Z    +0.000, E1   +49.801, E3 +325331.437}
SPL {X  -162.820, Y  +386.334, Z    +0.000, E1   +49.739, E3 +325341.525}
SPL {X  -162.801, Y  +377.981, Z    +0.000, E1   +49.798, E3 +325356.047}
SPL {X  -162.314, Y  +367.677, Z    +0.000, E1   +49.734, E3 +325374.686}
SPL {X  -161.614, Y  +360.718, Z    +0.000, E1   +49.491, E3 +325388.104}
SPL {X  -160.828, Y  +355.106, Z    +0.000, E1   +49.536, E3 +325397.788}
SPL {X  -159.832, Y  +349.452, Z    +0.000, E1   +49.188, E3 +325409.759}
SPL {X  -158.863, Y  +344.823, Z    +0.000, E1   +49.020, E3 +325418.808}
SPL {X  -157.695, Y  +339.971, Z    +0.000, E1   +48.934, E3 +325427.905}
SPL {X  -156.136, Y  +334.326, Z    +0.000, E1   +48.578, E3 +325439.871}
SPL {X  -154.561, Y  +329.302, Z    +0.000, E1   +48.290, E3 +325450.202}
SPL {X  -152.787, Y  +324.229, Z    +0.000, E1   +47.981, E3 +325460.892}
SPL {X  -150.789, Y  +319.074, Z    +0.000, E1   +47.585, E3 +325471.914}
SPL {X  -145.123, Y  +306.679, Z    +0.000, E1   +50.518, E3 +325477.812}
SPL {X  -135.207, Y  +289.783, Z    +0.000, E1   +44.101, E3 +325571.326}
ENDSPLINE

SPLINE
SPL {X  -154.528, Y  +329.203, Z    +0.000, E1   +28.834, E3 +325641.687}
SPL {X  -160.380, Y  +352.419, Z    +0.000, E1   +18.163, E3 +325646.048}
SPL {X  -162.408, Y  +368.921, Z    +0.000, E1    +9.337, E3 +325644.798}
SPL {X  -162.817, Y  +379.558, Z    +0.000, E1    +2.744, E3 +325645.188}
SPL {X  -162.820, Y  +383.077, Z    +0.000, E1    +0.110, E3 +325645.583}
SPL {X  -162.820, Y  +386.028, Z    +0.000, E1    -2.328, E3 +325644.906}
SPL {X  -162.820, Y  +389.792, Z    +0.000, E1    -6.211, E3 +325644.838}
SPL {X  -162.820, Y  +394.068, Z    +0.000, E1   -11.043, E3 +325644.955}
SPL {X  -162.820, Y  +398.921, Z    +0.000, E1   -16.945, E3 +325645.008}
SPL {X  -162.820, Y  +409.049, Z    +0.000, E1   -29.128, E3 +325643.817}
SPL {X  -162.820, Y  +444.592, Z    +0.000, E1   -49.032, E3 +325662.827}
SPL {X  -162.820, Y  +458.217, Z    +0.000, E1   -51.268, E3 +325674.772}
SPL {X  -162.820, Y  +501.848, Z    +0.000, E1   -54.235, E3 +325721.140}
ENDSPLINE

SPLINE
SPL {X  -162.820, Y  +498.156, Z    +0.000, E1   -50.986, E3 +325734.689}
ENDSPLINE

SPLINE
SPL {X  -162.820, Y  +499.429, Z    +0.000, E1   -49.453, E3 +325746.048}
SPL {X  -162.820, Y  +505.173, Z    +0.000, E1   -49.386, E3 +325756.703}
SPL {X  -162.820, Y  +510.642, Z    +0.000, E1   -49.447, E3 +325766.053}
SPL {X  -162.820, Y  +516.435, Z    +0.000, E1   -49.526, E3 +325775.931}
SPL {X  -162.820, Y  +522.095, Z    +0.000, E1   -49.420, E3 +325786.628}
SPL {X  -162.820, Y  +529.397, Z    +0.000, E1   -49.440, E3 +325799.637}
SPL {X  -162.820, Y  +536.932, Z    +0.000, E1   -49.395, E3 +325813.278}
SPL {X  -162.820, Y  +543.021, Z    +0.000, E1   -49.432, E3 +325823.884}
SPL {X  -162.820, Y  +548.933, Z    +0.000, E1   -49.456, E3 +325834.287}
SPL {X  -162.820, Y  +553.997, Z    +0.000, E1   -49.325, E3 +325844.091}
SPL {X  -162.820, Y  +562.346, Z    +0.000, E1   -49.498, E3 +325858.154}
SPL {X  -162.820, Y  +570.444, Z    +0.000, E1   -49.421, E3 +325872.900}
SPL {X  -162.820, Y  +577.429, Z    +0.000, E1   -49.474, E3 +325885.015}
SPL {X  -162.820, Y  +585.965, Z    +0.000, E1   -49.447, E3 +325900.588}
SPL {X  -162.820, Y  +594.192, Z    +0.000, E1   -49.325, E3 +325915.832}
SPL {X  -162.820, Y  +600.267, Z    +0.000, E1   -49.443, E3 +325925.920}
SPL {X  -162.820, Y  +606.218, Z    +0.000, E1   -49.464, E3 +325936.467}
SPL {X  -162.820, Y  +612.538, Z    +0.000, E1   -49.488, E3 +325947.518}
SPL {X  -162.820, Y  +617.738, Z    +0.000, E1   -49.301, E3 +325957.954}
SPL {X  -162.820, Y  +624.265, Z    +0.000, E1   -49.443, E3 +325968.750}
SPL {X  -162.820, Y  +632.551, Z    +0.000, E1   -49.478, E3 +325983.518}
SPL {X  -162.820, Y  +641.207, Z    +0.000, E1   -49.420, E3 +325999.162}
SPL {X  -162.820, Y  +648.011, Z    +0.000, E1   -49.484, E3 +326010.839}
SPL {X  -162.820, Y  +655.976, Z    +0.000, E1   -49.445, E3 +326025.467}
SPL {X  -162.820, Y  +663.916, Z    +0.000, E1   -49.371, E3 +326039.896}
SPL {X  -162.820, Y  +669.755, Z    +0.000, E1   -49.387, E3 +326050.221}
SPL {X  -162.807, Y  +675.597, Z    +0.000, E1   -49.472, E3 +326060.124}
SPL {X  -162.632, Y  +681.322, Z    +0.000, E1   -49.345, E3 +326071.135}
SPL {X  -162.228, Y  +687.372, Z    +0.000, E1   -49.294, E3 +326082.221}
SPL {X  -161.723, Y  +692.372, Z    +0.000, E1   -49.172, E3 +326091.852}
SPL {X  -161.009, Y  +697.714, Z    +0.000, E1   -49.214, E3 +326101.136}
SPL {X  -160.313, Y  +701.965, Z    +0.000, E1   -48.932, E3 +326110.348}
SPL {X  -158.980, Y  +708.651, Z    +0.000, E1   -48.774, E3 +326123.389}
SPL {X  -157.477, Y  +714.869, Z    +0.000, E1   -48.424, E3 +326136.263}
SPL {X  -156.071, Y  +719.891, Z    +0.000, E1   -48.264, E3 +326146.140}
SPL {X  -154.661, Y  +724.395, Z    +0.000, E1   -47.951, E3 +326155.821}
SPL {X  -153.094, Y  +728.931, Z    +0.000, E1   -47.705, E3 +326165.258}
SPL {X  -151.300, Y  +733.655, Z    +0.000, E1   -47.339, E3 +326175.566}
SPL {X  -145.669, Y  +746.239, Z    +0.000, E1   -50.198, E3 +326182.343}
SPL {X  -135.084, Y  +764.399, Z    +0.000, E1   -44.787, E3 +326265.247}
ENDSPLINE

SPLINE
SPL {X  -153.038, Y  +729.086, Z    +0.000, E1   -30.522, E3 +326335.953}
SPL {X  -160.383, Y  +701.564, Z    +0.000, E1   -18.145, E3 +326345.990}
SPL {X  -162.078, Y  +689.023, Z    +0.000, E1   -11.510, E3 +326345.528}
SPL {X  -162.685, Y  +680.136, Z    +0.000, E1    -6.379, E3 +326345.816}
SPL {X  -162.814, Y  +674.937, Z    +0.000, E1    -3.051, E3 +326345.886}
SPL {X  -162.820, Y  +671.865, Z    +0.000, E1    -0.918, E3 +326345.837}
SPL {X  -162.820, Y  +667.861, Z    +0.000, E1    +2.254, E3 +326345.656}
SPL {X  -162.820, Y  +662.755, Z    +0.000, E1    +7.521, E3 +326345.697}
SPL {X  -162.820, Y  +657.537, Z    +0.000, E1   +13.540, E3 +326345.366}
SPL {X  -162.820, Y  +650.460, Z    +0.000, E1   +22.200, E3 +326344.797}
SPL {X  -162.820, Y  +637.843, Z    +0.000, E1   +35.051, E3 +326346.874}
SPL {X  -162.820, Y  +595.072, Z    +0.000, E1   +53.652, E3 +326367.594}
SPL {X  -162.820, Y  +560.706, Z    +0.000, E1   +50.482, E3 +326428.503}
ENDSPLINE

SPLINE
SPL {X  -162.820, Y  +560.978, Z    +0.000, E1   +48.448, E3 +326440.589}
ENDSPLINE

SPLINE
SPL {X  -162.820, Y  +552.125, Z    +0.000, E1   +48.477, E3 +326456.694}
SPL {X  -162.820, Y  +545.800, Z    +0.000, E1   +48.334, E3 +326469.136}
SPL {X  -162.820, Y  +540.645, Z    +0.000, E1   +48.364, E3 +326478.486}
SPL {X  -162.820, Y  +534.689, Z    +0.000, E1   +48.295, E3 +326490.035}
SPL {X  -162.820, Y  +526.053, Z    +0.000, E1   +48.382, E3 +326505.610}
SPL {X  -162.820, Y  +519.666, Z    +0.000, E1   +48.261, E3 +326517.979}
SPL {X  -162.820, Y  +512.600, Z    +0.000, E1   +48.469, E3 +326529.965}
SPL {X  -162.820, Y  +504.728, Z    +0.000, E1   +48.342, E3 +326545.294}
ENDSPLINE

SPLINE
SPL {X  -162.820, Y  +517.326, Z    +0.000, E1   +41.232, E3 +326561.014}
ENDSPLINE

SPLINE
SPL {X  -162.820, Y  +507.007, Z    +0.000, E1   +42.470, E3 +326577.692}
SPL {X  -162.820, Y  +496.780, Z    +0.000, E1   +43.573, E3 +326593.947}
SPL {X  -162.820, Y  +488.962, Z    +0.000, E1   +44.342, E3 +326606.215}
SPL {X  -162.820, Y  +481.373, Z    +0.000, E1   +45.107, E3 +326617.699}
SPL {X  -162.820, Y  +473.909, Z    +0.000, E1   +45.743, E3 +326629.212}
SPL {X  -162.820, Y  +463.464, Z    +0.000, E1   +47.025, E3 +326642.429}
SPL {X  -162.820, Y  +451.336, Z    +0.000, E1   +48.248, E3 +326658.199}
SPL {X  -162.820, Y  +440.303, Z    +0.000, E1   +49.204, E3 +326672.646}
SPL {X  -162.820, Y  +430.072, Z    +0.000, E1   +49.865, E3 +326686.948}
SPL {X  -162.820, Y  +423.062, Z    +0.000, E1   +49.728, E3 +326699.942}
SPL {X  -162.820, Y  +416.560, Z    +0.000, E1   +49.816, E3 +326710.923}
SPL {X  -162.820, Y  +410.559, Z    +0.000, E1   +49.727, E3 +326721.978}
SPL {X  -162.820, Y  +402.501, Z    +0.000, E1   +49.838, E3 +326735.667}
SPL {X  -162.820, Y  +393.582, Z    +0.000, E1   +49.779, E3 +326751.664}
SPL {X  -162.820, Y  +386.334, Z    +0.000, E1   +49.739, E3 +326764.602}
SPL {X  -162.820, Y  +381.297, Z    +0.000, E1   +49.665, E3 +326773.873}
SPL {X  -162.709, Y  +374.487, Z    +0.000, E1   +49.773, E3 +326785.398}
SPL {X  -162.299, Y  +367.483, Z    +0.000, E1   +49.784, E3 +326797.540}
SPL {X  -161.760, Y  +361.947, Z    +0.000, E1   +49.515, E3 +326808.948}
SPL {X  -160.828, Y  +355.106, Z    +0.000, E1   +49.536, E3 +326820.865}
SPL {X  -159.832, Y  +349.452, Z    +0.000, E1   +49.188, E3 +326832.836}
SPL {X  -158.863, Y  +344.823, Z    +0.000, E1   +49.020, E3 +326841.885}
SPL {X  -157.695, Y  +339.971, Z    +0.000, E1   +48.934, E3 +326850.982}
SPL {X  -156.496, Y  +335.563, Z    +0.000, E1   +48.599, E3 +326860.559}
SPL {X  -154.894, Y  +330.318, Z    +0.000, E1   +48.380, E3 +326871.102}
SPL {X  -153.352, Y  +325.786, Z    +0.000, E1   +48.028, E3 +326880.858}
SPL {X  -151.316, Y  +320.384, Z    +0.000, E1   +47.734, E3 +326892.074}
SPL {X  -145.123, Y  +306.679, Z    +0.000, E1   +50.518, E3 +326900.889}
SPL {X  -135.207, Y  +289.783, Z    +0.000, E1   +44.101, E3 +326994.403}
ENDSPLINE

SPLINE
SPL {X  -154.528, Y  +329.203, Z    +0.000, E1   +28.834, E3 +327064.764}
SPL {X  -160.380, Y  +352.419, Z    +0.000, E1   +18.163, E3 +327069.125}
SPL {X  -162.149, Y  +365.734, Z    +0.000, E1   +11.090, E3 +327067.733}
SPL {X  -162.754, Y  +375.862, Z    +0.000, E1    +5.134, E3 +327068.570}
SPL {X  -162.820, Y  +382.085, Z    +0.000, E1    +0.928, E3 +327068.259}
SPL {X  -162.820, Y  +386.028, Z    +0.000, E1    -2.328, E3 +327067.983}
SPL {X  -162.820, Y  +389.792, Z    +0.000, E1    -6.211, E3 +327067.915}
SPL {X  -162.820, Y  +394.068, Z    +0.000, E1   -11.043, E3 +327068.032}
SPL {X  -162.820, Y  +398.921, Z    +0.000, E1   -16.945, E3 +327068.085}
SPL {X  -162.820, Y  +409.049, Z    +0.000, E1   -29.128, E3 +327066.894}
SPL {X  -162.820, Y  +446.299, Z    +0.000, E1   -49.360, E3 +327087.398}
SPL {X  -162.820, Y  +502.427, Z    +0.000, E1   -53.345, E3 +327150.383}
ENDSPLINE

SPLINE
SPL {X  -162.820, Y  +494.458, Z    +0.000, E1   -49.332, E3 +327160.915}
ENDSPLINE

SPLINE
SPL {X  -162.820, Y  +499.429, Z    +0.000, E1   -49.453, E3 +327169.125}
SPL {X  -162.820, Y  +507.703, Z    +0.000, E1   -49.462, E3 +327184.040}
SPL {X  -162.820, Y  +516.435, Z    +0.000, E1   -49.526, E3 +327199.008}
SPL {X  -162.820, Y  +522.095, Z    +0.000, E1   -49.420, E3 +327209.705}
SPL {X  -162.820, Y  +529.397, Z    +0.000, E1   -49.440, E3 +327222.714}
SPL {X  -162.820, Y  +535.099, Z    +0.000, E1   -49.339, E3 +327233.332}
SPL {X  -162.820, Y  +541.471, Z    +0.000, E1   -49.456, E3 +327244.176}
SPL {X  -162.820, Y  +548.933, Z    +0.000, E1   -49.456, E3 +327257.364}
SPL {X  -162.820, Y  +553.997, Z    +0.000, E1   -49.325, E3 +327267.168}
SPL {X  -162.820, Y  +560.268, Z    +0.000, E1   -49.531, E3 +327277.126}
SPL {X  -162.820, Y  +564.590, Z    +0.000, E1   -49.361, E3 +327285.826}
SPL {X  -162.820, Y  +570.444, Z    +0.000, E1   -49.421, E3 +327295.977}
SPL {X  -162.820, Y  +577.429, Z    +0.000, E1   -49.474, E3 +327308.092}
SPL {X  -162.820, Y  +582.387, Z    +0.000, E1   -49.269, E3 +327318.113}
SPL {X  -162.820, Y  +588.456, Z    +0.000, E1   -49.496, E3 +327327.627}
SPL {X  -162.820, Y  +594.192, Z    +0.000, E1   -49.325, E3 +327338.908}
SPL {X  -162.820, Y  +600.267, Z    +0.000, E1   -49.443, E3 +327348.997}
SPL {X  -162.820, Y  +606.218, Z    +0.000, E1   -49.464, E3 +327359.544}
SPL {X  -162.820, Y  +612.538, Z    +0.000, E1   -49.488, E3 +327370.595}
SPL {X  -162.820, Y  +617.738, Z    +0.000, E1   -49.301, E3 +327381.031}
SPL {X  -162.820, Y  +624.265, Z    +0.000, E1   -49.443, E3 +327391.826}
SPL {X  -162.820, Y  +630.226, Z    +0.000, E1   -49.472, E3 +327402.275}
SPL {X  -162.820, Y  +635.239, Z    +0.000, E1   -49.373, E3 +327411.770}
SPL {X  -162.820, Y  +641.207, Z    +0.000, E1   -49.420, E3 +327422.238}
SPL {X  -162.820, Y  +649.864, Z    +0.000, E1   -49.433, E3 +327437.717}
SPL {X  -162.820, Y  +658.147, Z    +0.000, E1   -49.491, E3 +327451.984}
SPL {X  -162.820, Y  +663.916, Z    +0.000, E1   -49.371, E3 +327462.973}
SPL {X  -162.820, Y  +669.755, Z    +0.000, E1   -49.387, E3 +327473.298}
SPL {X  -162.807, Y  +675.597, Z    +0.000, E1   -49.472, E3 +327483.201}
SPL {X  -162.632, Y  +681.322, Z    +0.000, E1   -49.345, E3 +327494.212}
SPL {X  -162.228, Y  +687.372, Z    +0.000, E1   -49.294, E3 +327505.298}
SPL {X  -161.723, Y  +692.372, Z    +0.000, E1   -49.172, E3 +327514.929}
SPL {X  -161.009, Y  +697.714, Z    +0.000, E1   -49.214, E3 +327524.213}
SPL {X  -160.313, Y  +701.965, Z    +0.000, E1   -48.932, E3 +327533.425}
SPL {X  -159.435, Y  +706.528, Z    +0.000, E1   -48.764, E3 +327542.552}
SPL {X  -157.894, Y  +713.249, Z    +0.000, E1   -48.586, E3 +327555.746}
SPL {X  -156.071, Y  +719.891, Z    +0.000, E1   -48.264, E3 +327569.217}
SPL {X  -154.661, Y  +724.395, Z    +0.000, E1   -47.951, E3 +327578.898}
SPL {X  -153.094, Y  +728.931, Z    +0.000, E1   -47.705, E3 +327588.335}
SPL {X  -151.300, Y  +733.655, Z    +0.000, E1   -47.339, E3 +327598.643}
SPL {X  -145.669, Y  +746.239, Z    +0.000, E1   -50.198, E3 +327605.420}
SPL {X  -135.084, Y  +764.399, Z    +0.000, E1   -44.787, E3 +327688.324}
ENDSPLINE

SPLINE
SPL {X  -153.038, Y  +729.086, Z    +0.000, E1   -30.522, E3 +327759.030}
SPL {X  -160.383, Y  +701.564, Z    +0.000, E1   -18.145, E3 +327769.066}
SPL {X  -162.078, Y  +689.023, Z    +0.000, E1   -11.510, E3 +327768.604}
SPL {X  -162.685, Y  +680.136, Z    +0.000, E1    -6.379, E3 +327768.893}
SPL {X  -162.820, Y  +672.919, Z    +0.000, E1    -1.752, E3 +327768.932}
SPL {X  -162.820, Y  +669.270, Z    +0.000, E1    +1.140, E3 +327768.414}
SPL {X  -162.820, Y  +666.754, Z    +0.000, E1    +3.396, E3 +327768.984}
SPL {X  -162.820, Y  +662.755, Z    +0.000, E1    +7.521, E3 +327768.774}
SPL {X  -162.820, Y  +657.537, Z    +0.000, E1   +13.540, E3 +327768.443}
SPL {X  -162.820, Y  +650.460, Z    +0.000, E1   +22.200, E3 +327767.874}
SPL {X  -162.820, Y  +637.843, Z    +0.000, E1   +35.051, E3 +327769.951}
SPL {X  -162.820, Y  +595.072, Z    +0.000, E1   +53.652, E3 +327790.671}
SPL {X  -162.820, Y  +561.831, Z    +0.000, E1   +49.171, E3 +327857.894}
SPL {X  -162.820, Y  +555.289, Z    +0.000, E1   +48.406, E3 +327874.355}
SPL {X  -162.820, Y  +547.003, Z    +0.000, E1   +48.390, E3 +327889.767}
SPL {X  -162.820, Y  +540.645, Z    +0.000, E1   +48.364, E3 +327901.563}
SPL {X  -162.820, Y  +534.689, Z    +0.000, E1   +48.295, E3 +327913.112}
SPL {X  -162.820, Y  +526.053, Z    +0.000, E1   +48.382, E3 +327928.687}
SPL {X  -162.820, Y  +519.666, Z    +0.000, E1   +48.261, E3 +327941.056}
SPL {X  -162.820, Y  +512.600, Z    +0.000, E1   +48.469, E3 +327953.042}
SPL {X  -162.820, Y  +504.728, Z    +0.000, E1   +48.342, E3 +327968.371}
ENDSPLINE

SPLINE
SPL {X  -162.820, Y  +517.326, Z    +0.000, E1   +41.232, E3 +327984.091}
ENDSPLINE

SPLINE
SPL {X  -162.820, Y  +507.007, Z    +0.000, E1   +42.470, E3 +328000.769}
SPL {X  -162.820, Y  +496.780, Z    +0.000, E1   +43.573, E3 +328017.024}
SPL {X  -162.820, Y  +488.962, Z    +0.000, E1   +44.342, E3 +328029.292}
SPL {X  -162.820, Y  +481.373, Z    +0.000, E1   +45.107, E3 +328040.776}
SPL {X  -162.820, Y  +473.909, Z    +0.000, E1   +45.743, E3 +328052.289}
SPL {X  -162.820, Y  +465.836, Z    +0.000, E1   +46.727, E3 +328062.580}
SPL {X  -162.820, Y  +457.217, Z    +0.000, E1   +47.671, E3 +328073.618}
SPL {X  -162.820, Y  +449.104, Z    +0.000, E1   +48.459, E3 +328084.086}
SPL {X  -162.820, Y  +440.303, Z    +0.000, E1   +49.204, E3 +328095.723}
SPL {X  -162.820, Y  +430.072, Z    +0.000, E1   +49.865, E3 +328110.025}
SPL {X  -162.820, Y  +423.062, Z    +0.000, E1   +49.728, E3 +328123.019}
SPL {X  -162.820, Y  +416.560, Z    +0.000, E1   +49.816, E3 +328134.000}
SPL {X  -162.820, Y  +410.559, Z    +0.000, E1   +49.727, E3 +328145.055}
SPL {X  -162.820, Y  +405.170, Z    +0.000, E1   +49.772, E3 +328154.257}
SPL {X  -162.820, Y  +398.766, Z    +0.000, E1   +49.793, E3 +328165.545}
SPL {X  -162.820, Y  +391.831, Z    +0.000, E1   +49.801, E3 +328177.590}
SPL {X  -162.820, Y  +386.334, Z    +0.000, E1   +49.739, E3 +328187.679}
SPL {X  -162.801, Y  +377.981, Z    +0.000, E1   +49.798, E3 +328202.201}
SPL {X  -162.314, Y  +367.677, Z    +0.000, E1   +49.734, E3 +328220.840}
SPL {X  -161.614, Y  +360.718, Z    +0.000, E1   +49.491, E3 +328234.258}
SPL {X  -160.828, Y  +355.106, Z    +0.000, E1   +49.536, E3 +328243.942}
SPL {X  -159.832, Y  +349.452, Z    +0.000, E1   +49.188, E3 +328255.913}
SPL {X  -158.863, Y  +344.823, Z    +0.000, E1   +49.020, E3 +328264.962}
SPL {X  -157.695, Y  +339.971, Z    +0.000, E1   +48.934, E3 +328274.059}
SPL {X  -156.496, Y  +335.563, Z    +0.000, E1   +48.599, E3 +328283.636}
SPL {X  -154.894, Y  +330.318, Z    +0.000, E1   +48.380, E3 +328294.179}
SPL {X  -153.352, Y  +325.786, Z    +0.000, E1   +48.028, E3 +328303.935}
SPL {X  -151.655, Y  +321.245, Z    +0.000, E1   +47.770, E3 +328313.356}
SPL {X  -148.347, Y  +313.391, Z    +0.000, E1   +48.924, E3 +328320.954}
SPL {X  -143.047, Y  +302.732, Z    +0.000, E1   +51.043, E3 +328327.474}
SPL {X  -134.119, Y  +288.184, Z    +0.000, E1   +45.142, E3 +328407.369}
ENDSPLINE

SPLINE
SPL {X  -136.325, Y  +291.473, Z    +0.000, E1   +43.106, E3 +328425.945}
SPL {X  -154.528, Y  +329.203, Z    +0.000, E1   +28.834, E3 +328487.841}
SPL {X  -160.380, Y  +352.419, Z    +0.000, E1   +18.163, E3 +328492.202}
SPL {X  -162.149, Y  +365.734, Z    +0.000, E1   +11.090, E3 +328490.810}
SPL {X  -162.754, Y  +375.862, Z    +0.000, E1    +5.134, E3 +328491.647}
SPL {X  -162.820, Y  +382.085, Z    +0.000, E1    +0.928, E3 +328491.336}
SPL {X  -162.820, Y  +386.028, Z    +0.000, E1    -2.328, E3 +328491.060}
SPL {X  -162.820, Y  +389.792, Z    +0.000, E1    -6.211, E3 +328490.992}
SPL {X  -162.820, Y  +394.068, Z    +0.000, E1   -11.043, E3 +328491.109}
SPL {X  -162.820, Y  +398.921, Z    +0.000, E1   -16.945, E3 +328491.162}
SPL {X  -162.820, Y  +409.049, Z    +0.000, E1   -29.128, E3 +328489.971}
SPL {X  -162.820, Y  +444.592, Z    +0.000, E1   -49.032, E3 +328508.981}
SPL {X  -162.820, Y  +458.217, Z    +0.000, E1   -51.268, E3 +328520.926}
SPL {X  -162.820, Y  +501.848, Z    +0.000, E1   -54.235, E3 +328567.294}
ENDSPLINE

SPLINE
SPL {X  -162.820, Y  +498.156, Z    +0.000, E1   -50.986, E3 +328580.843}
ENDSPLINE

SPLINE
SPL {X  -162.820, Y  +499.429, Z    +0.000, E1   -49.453, E3 +328592.202}
SPL {X  -162.820, Y  +505.173, Z    +0.000, E1   -49.386, E3 +328602.857}
SPL {X  -162.820, Y  +510.642, Z    +0.000, E1   -49.447, E3 +328612.207}
SPL {X  -162.820, Y  +516.435, Z    +0.000, E1   -49.526, E3 +328622.085}
SPL {X  -162.820, Y  +522.095, Z    +0.000, E1   -49.420, E3 +328632.782}
SPL {X  -162.820, Y  +529.397, Z    +0.000, E1   -49.440, E3 +328645.791}
SPL {X  -162.820, Y  +536.932, Z    +0.000, E1   -49.395, E3 +328659.432}
SPL {X  -162.820, Y  +543.021, Z    +0.000, E1   -49.432, E3 +328670.038}
SPL {X  -162.820, Y  +548.933, Z    +0.000, E1   -49.456, E3 +328680.441}
SPL {X  -162.820, Y  +553.997, Z    +0.000, E1   -49.325, E3 +328690.245}
SPL {X  -162.820, Y  +562.346, Z    +0.000, E1   -49.498, E3 +328704.307}
SPL {X  -162.820, Y  +570.444, Z    +0.000, E1   -49.421, E3 +328719.054}
SPL {X  -162.820, Y  +577.429, Z    +0.000, E1   -49.474, E3 +328731.168}
SPL {X  -162.820, Y  +585.965, Z    +0.000, E1   -49.447, E3 +328746.742}
SPL {X  -162.820, Y  +594.192, Z    +0.000, E1   -49.325, E3 +328761.985}
SPL {X  -162.820, Y  +600.267, Z    +0.000, E1   -49.443, E3 +328772.074}
SPL {X  -162.820, Y  +606.218, Z    +0.000, E1   -49.464, E3 +328782.621}
SPL {X  -162.820, Y  +612.538, Z    +0.000, E1   -49.488, E3 +328793.672}
SPL {X  -162.820, Y  +617.738, Z    +0.000, E1   -49.301, E3 +328804.108}
SPL {X  -162.820, Y  +624.265, Z    +0.000, E1   -49.443, E3 +328814.903}
SPL {X  -162.820, Y  +632.551, Z    +0.000, E1   -49.478, E3 +328829.672}
SPL {X  -162.820, Y  +641.207, Z    +0.000, E1   -49.420, E3 +328845.315}
SPL {X  -162.820, Y  +648.011, Z    +0.000, E1   -49.484, E3 +328856.992}
SPL {X  -162.820, Y  +655.976, Z    +0.000, E1   -49.445, E3 +328871.621}
SPL {X  -162.820, Y  +663.916, Z    +0.000, E1   -49.371, E3 +328886.050}
SPL {X  -162.820, Y  +669.755, Z    +0.000, E1   -49.387, E3 +328896.375}
SPL {X  -162.807, Y  +675.597, Z    +0.000, E1   -49.472, E3 +328906.277}
SPL {X  -162.632, Y  +681.322, Z    +0.000, E1   -49.345, E3 +328917.289}
SPL {X  -162.228, Y  +687.372, Z    +0.000, E1   -49.294, E3 +328928.375}
SPL {X  -161.723, Y  +692.372, Z    +0.000, E1   -49.172, E3 +328938.006}
SPL {X  -161.009, Y  +697.714, Z    +0.000, E1   -49.214, E3 +328947.290}
SPL {X  -160.313, Y  +701.965, Z    +0.000, E1   -48.932, E3 +328956.502}
SPL {X  -159.435, Y  +706.528, Z    +0.000, E1   -48.764, E3 +328965.629}
SPL {X  -157.894, Y  +713.249, Z    +0.000, E1   -48.586, E3 +328978.823}
SPL {X  -156.071, Y  +719.891, Z    +0.000, E1   -48.264, E3 +328992.294}
SPL {X  -154.661, Y  +724.395, Z    +0.000, E1   -47.951, E3 +329001.975}
SPL {X  -153.094, Y  +728.931, Z    +0.000, E1   -47.705, E3 +329011.412}
SPL {X  -151.300, Y  +733.655, Z    +0.000, E1   -47.339, E3 +329021.720}
SPL {X  -145.669, Y  +746.239, Z    +0.000, E1   -50.198, E3 +329028.497}
SPL {X  -135.084, Y  +764.399, Z    +0.000, E1   -44.787, E3 +329111.400}
ENDSPLINE

SPLINE
SPL {X  -153.038, Y  +729.086, Z    +0.000, E1   -30.522, E3 +329182.107}
SPL {X  -160.383, Y  +701.564, Z    +0.000, E1   -18.145, E3 +329192.143}
SPL {X  -162.078, Y  +689.023, Z    +0.000, E1   -11.510, E3 +329191.681}
SPL {X  -162.685, Y  +680.136, Z    +0.000, E1    -6.379, E3 +329191.970}
SPL {X  -162.820, Y  +672.919, Z    +0.000, E1    -1.752, E3 +329192.009}
SPL {X  -162.820, Y  +667.861, Z    +0.000, E1    +2.254, E3 +329191.810}
SPL {X  -162.820, Y  +662.755, Z    +0.000, E1    +7.521, E3 +329191.851}
SPL {X  -162.820, Y  +657.537, Z    +0.000, E1   +13.540, E3 +329191.520}
SPL {X  -162.820, Y  +650.460, Z    +0.000, E1   +22.200, E3 +329190.951}
SPL {X  -162.820, Y  +637.843, Z    +0.000, E1   +35.051, E3 +329193.028}
SPL {X  -162.820, Y  +595.072, Z    +0.000, E1   +53.652, E3 +329213.748}
SPL {X  -162.820, Y  +561.831, Z    +0.000, E1   +49.171, E3 +329280.971}
SPL {X  -162.820, Y  +555.289, Z    +0.000, E1   +48.406, E3 +329297.432}
SPL {X  -162.820, Y  +547.003, Z    +0.000, E1   +48.390, E3 +329312.844}
SPL {X  -162.820, Y  +538.900, Z    +0.000, E1   +48.334, E3 +329328.204}
SPL {X  -162.820, Y  +530.572, Z    +0.000, E1   +48.392, E3 +329343.255}
SPL {X  -162.820, Y  +524.414, Z    +0.000, E1   +48.297, E3 +329355.137}
SPL {X  -162.820, Y  +519.666, Z    +0.000, E1   +48.261, E3 +329364.133}
SPL {X  -162.820, Y  +512.600, Z    +0.000, E1   +48.469, E3 +329376.119}
SPL {X  -162.820, Y  +504.728, Z    +0.000, E1   +48.342, E3 +329391.448}
ENDSPLINE

SPLINE
SPL {X  -162.820, Y  +520.386, Z    +0.000, E1   +40.911, E3 +329401.634}
ENDSPLINE

SPLINE
SPL {X  -162.820, Y  +515.876, Z    +0.000, E1   +41.348, E3 +329409.832}
SPL {X  -162.820, Y  +507.007, Z    +0.000, E1   +42.470, E3 +329423.846}
SPL {X  -162.820, Y  +496.780, Z    +0.000, E1   +43.573, E3 +329440.101}
SPL {X  -162.820, Y  +488.962, Z    +0.000, E1   +44.342, E3 +329452.369}
SPL {X  -162.820, Y  +481.373, Z    +0.000, E1   +45.107, E3 +329463.853}
SPL {X  -162.820, Y  +473.909, Z    +0.000, E1   +45.743, E3 +329475.366}
SPL {X  -162.820, Y  +465.836, Z    +0.000, E1   +46.727, E3 +329485.657}
SPL {X  -162.820, Y  +457.217, Z    +0.000, E1   +47.671, E3 +329496.695}
SPL {X  -162.820, Y  +449.104, Z    +0.000, E1   +48.459, E3 +329507.163}
SPL {X  -162.820, Y  +440.303, Z    +0.000, E1   +49.204, E3 +329518.800}
SPL {X  -162.820, Y  +430.072, Z    +0.000, E1   +49.865, E3 +329533.102}
SPL {X  -162.820, Y  +423.062, Z    +0.000, E1   +49.728, E3 +329546.096}
SPL {X  -162.820, Y  +416.560, Z    +0.000, E1   +49.816, E3 +329557.077}
SPL {X  -162.820, Y  +410.559, Z    +0.000, E1   +49.727, E3 +329568.132}
SPL {X  -162.820, Y  +405.170, Z    +0.000, E1   +49.772, E3 +329577.334}
SPL {X  -162.820, Y  +398.766, Z    +0.000, E1   +49.793, E3 +329588.621}
SPL {X  -162.820, Y  +391.831, Z    +0.000, E1   +49.801, E3 +329600.667}
SPL {X  -162.820, Y  +384.205, Z    +0.000, E1   +49.756, E3 +329614.599}
SPL {X  -162.753, Y  +375.844, Z    +0.000, E1   +49.816, E3 +329628.775}
SPL {X  -162.415, Y  +369.029, Z    +0.000, E1   +49.751, E3 +329641.264}
SPL {X  -161.760, Y  +361.947, Z    +0.000, E1   +49.515, E3 +329655.102}
SPL {X  -161.057, Y  +356.607, Z    +0.000, E1   +49.516, E3 +329664.414}
SPL {X  -160.051, Y  +350.597, Z    +0.000, E1   +49.332, E3 +329676.311}
SPL {X  -158.863, Y  +344.823, Z    +0.000, E1   +49.020, E3 +329688.039}
SPL {X  -157.695, Y  +339.971, Z    +0.000, E1   +48.934, E3 +329697.135}
SPL {X  -156.496, Y  +335.563, Z    +0.000, E1   +48.599, E3 +329706.713}
SPL {X  -154.894, Y  +330.318, Z    +0.000, E1   +48.380, E3 +329717.256}
SPL {X  -153.352, Y  +325.786, Z    +0.000, E1   +48.028, E3 +329727.012}
SPL {X  -151.316, Y  +320.384, Z    +0.000, E1   +47.734, E3 +329738.228}
SPL {X  -145.123, Y  +306.679, Z    +0.000, E1   +50.518, E3 +329747.043}
SPL {X  -135.207, Y  +289.783, Z    +0.000, E1   +44.101, E3 +329840.557}
ENDSPLINE

SPLINE
SPL {X  -154.528, Y  +329.203, Z    +0.000, E1   +28.834, E3 +329910.918}
SPL {X  -160.380, Y  +352.419, Z    +0.000, E1   +18.163, E3 +329915.278}
SPL {X  -162.149, Y  +365.734, Z    +0.000, E1   +11.090, E3 +329913.887}
SPL {X  -162.754, Y  +375.862, Z    +0.000, E1    +5.134, E3 +329914.724}
SPL {X  -162.820, Y  +382.085, Z    +0.000, E1    +0.928, E3 +329914.413}
SPL {X  -162.820, Y  +385.149, Z    +0.000, E1    -1.602, E3 +329914.139}
SPL {X  -162.820, Y  +388.871, Z    +0.000, E1    -5.151, E3 +329914.094}
SPL {X  -162.820, Y  +395.861, Z    +0.000, E1   -13.028, E3 +329914.205}
SPL {X  -162.820, Y  +409.049, Z    +0.000, E1   -29.128, E3 +329913.048}
SPL {X  -162.820, Y  +446.299, Z    +0.000, E1   -49.360, E3 +329933.552}
SPL {X  -162.820, Y  +502.427, Z    +0.000, E1   -53.345, E3 +329996.537}
ENDSPLINE

SPLINE
SPL {X  -162.820, Y  +494.458, Z    +0.000, E1   -49.332, E3 +330007.069}
ENDSPLINE

SPLINE
SPL {X  -162.820, Y  +499.429, Z    +0.000, E1   -49.453, E3 +330015.279}
SPL {X  -162.820, Y  +507.703, Z    +0.000, E1   -49.462, E3 +330030.193}
SPL {X  -162.820, Y  +516.435, Z    +0.000, E1   -49.526, E3 +330045.162}
SPL {X  -162.820, Y  +522.095, Z    +0.000, E1   -49.420, E3 +330055.859}
SPL {X  -162.820, Y  +529.397, Z    +0.000, E1   -49.440, E3 +330068.868}
SPL {X  -162.820, Y  +536.932, Z    +0.000, E1   -49.395, E3 +330082.508}
SPL {X  -162.820, Y  +543.021, Z    +0.000, E1   -49.432, E3 +330093.114}
SPL {X  -162.820, Y  +548.933, Z    +0.000, E1   -49.456, E3 +330103.518}
SPL {X  -162.820, Y  +553.997, Z    +0.000, E1   -49.325, E3 +330113.322}
SPL {X  -162.820, Y  +562.346, Z    +0.000, E1   -49.498, E3 +330127.384}
SPL {X  -162.820, Y  +570.444, Z    +0.000, E1   -49.421, E3 +330142.131}
SPL {X  -162.820, Y  +577.429, Z    +0.000, E1   -49.474, E3 +330154.245}
SPL {X  -162.820, Y  +582.387, Z    +0.000, E1   -49.269, E3 +330164.267}
SPL {X  -162.820, Y  +588.456, Z    +0.000, E1   -49.496, E3 +330173.781}
SPL {X  -162.820, Y  +594.192, Z    +0.000, E1   -49.325, E3 +330185.062}
SPL {X  -162.820, Y  +600.267, Z    +0.000, E1   -49.443, E3 +330195.151}
SPL {X  -162.820, Y  +606.218, Z    +0.000, E1   -49.464, E3 +330205.698}
SPL {X  -162.820, Y  +612.538, Z    +0.000, E1   -49.488, E3 +330216.749}
SPL {X  -162.820, Y  +617.738, Z    +0.000, E1   -49.301, E3 +330227.185}
SPL {X  -162.820, Y  +624.265, Z    +0.000, E1   -49.443, E3 +330237.980}
SPL {X  -162.820, Y  +632.551, Z    +0.000, E1   -49.478, E3 +330252.749}
SPL {X  -162.820, Y  +641.207, Z    +0.000, E1   -49.420, E3 +330268.392}
SPL {X  -162.820, Y  +649.864, Z    +0.000, E1   -49.433, E3 +330283.871}
SPL {X  -162.820, Y  +658.147, Z    +0.000, E1   -49.491, E3 +330298.137}
SPL {X  -162.820, Y  +663.916, Z    +0.000, E1   -49.371, E3 +330309.127}
SPL {X  -162.820, Y  +669.755, Z    +0.000, E1   -49.387, E3 +330319.452}
SPL {X  -162.807, Y  +675.597, Z    +0.000, E1   -49.472, E3 +330329.354}
SPL {X  -162.632, Y  +681.322, Z    +0.000, E1   -49.345, E3 +330340.366}
SPL {X  -162.228, Y  +687.372, Z    +0.000, E1   -49.294, E3 +330351.452}
SPL {X  -161.723, Y  +692.372, Z    +0.000, E1   -49.172, E3 +330361.083}
SPL {X  -161.009, Y  +697.714, Z    +0.000, E1   -49.214, E3 +330370.367}
SPL {X  -160.313, Y  +701.965, Z    +0.000, E1   -48.932, E3 +330379.579}
SPL {X  -158.980, Y  +708.651, Z    +0.000, E1   -48.774, E3 +330392.619}
SPL {X  -157.477, Y  +714.869, Z    +0.000, E1   -48.424, E3 +330405.494}
SPL {X  -156.071, Y  +719.891, Z    +0.000, E1   -48.264, E3 +330415.371}
SPL {X  -154.661, Y  +724.395, Z    +0.000, E1   -47.951, E3 +330425.052}
SPL {X  -153.094, Y  +728.931, Z    +0.000, E1   -47.705, E3 +330434.489}
SPL {X  -150.266, Y  +736.194, Z    +0.000, E1   -47.943, E3 +330446.097}
SPL {X  -143.458, Y  +750.508, Z    +0.000, E1   -51.034, E3 +330454.123}
SPL {X  -135.559, Y  +763.690, Z    +0.000, E1   -44.340, E3 +330538.368}
ENDSPLINE

SPLINE
SPL {X  -153.801, Y  +726.938, Z    +0.000, E1   -29.643, E3 +330607.081}
SPL {X  -160.383, Y  +701.564, Z    +0.000, E1   -18.145, E3 +330615.220}
SPL {X  -162.078, Y  +689.023, Z    +0.000, E1   -11.510, E3 +330614.758}
SPL {X  -162.685, Y  +680.136, Z    +0.000, E1    -6.379, E3 +330615.047}
SPL {X  -162.820, Y  +672.919, Z    +0.000, E1    -1.752, E3 +330615.086}
SPL {X  -162.820, Y  +667.861, Z    +0.000, E1    +2.254, E3 +330614.887}
SPL {X  -162.820, Y  +662.755, Z    +0.000, E1    +7.521, E3 +330614.928}
SPL {X  -162.820, Y  +657.537, Z    +0.000, E1   +13.540, E3 +330614.597}
SPL {X  -162.820, Y  +650.460, Z    +0.000, E1   +22.200, E3 +330614.028}
SPL {X  -162.820, Y  +637.843, Z    +0.000, E1   +35.051, E3 +330616.105}
SPL {X  -162.820, Y  +595.072, Z    +0.000, E1   +53.652, E3 +330636.825}
SPL {X  -162.820, Y  +560.706, Z    +0.000, E1   +50.482, E3 +330697.734}
ENDSPLINE

SPLINE
SPL {X  -162.820, Y  +560.978, Z    +0.000, E1   +48.448, E3 +330709.820}
ENDSPLINE

SPLINE
SPL {X  -162.820, Y  +552.125, Z    +0.000, E1   +48.477, E3 +330725.925}
SPL {X  -162.820, Y  +545.800, Z    +0.000, E1   +48.334, E3 +330738.366}
SPL {X  -162.820, Y  +538.900, Z    +0.000, E1   +48.334, E3 +330751.281}
SPL {X  -162.820, Y  +530.572, Z    +0.000, E1   +48.392, E3 +330766.332}
SPL {X  -162.820, Y  +522.157, Z    +0.000, E1   +48.326, E3 +330782.420}
SPL {X  -162.820, Y  +512.600, Z    +0.000, E1   +48.469, E3 +330799.196}
SPL {X  -162.820, Y  +504.728, Z    +0.000, E1   +48.342, E3 +330814.525}
ENDSPLINE

SPLINE
SPL {X  -162.820, Y  +517.326, Z    +0.000, E1   +41.232, E3 +330830.245}
ENDSPLINE

